                IF _sut_A._Step(_totalStepNumber - 1, TRUE, CONCAT('Step ', INT_TO_STRING(_totalStepNumber - 1))) THEN
                    _sut_A._SequenceComplete();
                END_IF

                _sut_A.SequencerClose();
                _sut_N.SequencerOpen();

                IF _sut_N._Step(0, TRUE, 'Step 0') THEN
                    _sut_N._StepCompleteWhen(TRUE);
                END_IF

                FOR i := 1 TO _totalStepNumber - 2 DO
                    _sut_N._Step(i, TRUE, CONCAT('Step ', INT_TO_STRING(i)));
                END_FOR

                IF _sut_N._Step(_totalStepNumber - 1, TRUE, CONCAT('Step ', INT_TO_STRING(_totalStepNumber - 1))) THEN
                    _sut_N._SequenceComplete();
                END_IF

                _sut_N.SequencerClose();
            END_IF

            IF _plcCycleCounter = 2 THEN
                _sut_A.SequencerOpen();

                IF _sut_A._Step(0, TRUE, 'Step 0') THEN
                    _sut_A._StepCompleteWhen(TRUE);
                END_IF

                IF _sut_A._Step(1, FALSE, 'Step 0') THEN
                    _sut_A._StepCompleteWhen(FALSE);
                END_IF

                _sut_N.SequencerOpen();

                IF _sut_N._Step(0, TRUE, 'Step 0') THEN
                    _sut_N._StepCompleteWhen(TRUE);
                END_IF

                IF _sut_N._Step(1, FALSE, 'Step 0') THEN
                    _sut_N._StepCompleteWhen(FALSE);
                END_IF
            END_IF

            IF _plcCycleCounter = 3 THEN
                FOR i := 2 TO _totalStepNumber - 1 DO
                    _sut_A._Step(i, TRUE, CONCAT('Step ', INT_TO_STRING(i)));
                END_FOR

                IF _sut_A._Step(_totalStepNumber, TRUE, CONCAT('Step ', INT_TO_STRING(_totalStepNumber))) THEN
                    _sut_A._SequenceComplete();
                END_IF

                _sut_A.SequencerClose();

                FOR i := 2 TO _totalStepNumber - 1 DO
                    _sut_N._Step(i, TRUE, CONCAT('Step ', INT_TO_STRING(i)));
                END_FOR

                IF _sut_N._Step(_totalStepNumber, TRUE, CONCAT('Step ', INT_TO_STRING(_totalStepNumber))) THEN
                    _sut_N._SequenceComplete();
                END_IF

                _sut_N.SequencerClose();
            END_IF

            _sut_A.SaveNumberOfStepsInSequence();
            _sut_N.SaveNumberOfStepsInSequence();
        END_IF

        _done := _plcCycleCounter >= 3;
        ProbeDoneWhen(_done);
        {endregion}
        {region "T560_RequestStepCallingCyclically"}
    eTcoSequencerTests.RequestStepCallingCyclically:
        IF NOT _arranged THEN
            _sut_A.TcoSequencerTest := eTcoSequencerTests.RequestStepCallingCyclically;
            _sut_N.TcoSequencerTest := eTcoSequencerTests.RequestStepCallingCyclically;
            _sut_A.SetCyclicMode(); //Set sequencer into the cyclic mode
            _sut_N.SetCyclicMode(); //Set sequencer into the cyclic mode
            _sut_A.SetSequenceAsChecked(); //Set sequence as checked, so no StepID uniqueness is performed on next sequence execution
            _sut_N.SetSequenceAsChecked(); //Set sequence as checked, so no StepID uniqueness is performed on next sequence execution
            _sut_A.SetNumberOfSteps(_totalStepNumber);
            _sut_N.SetNumberOfSteps(_totalStepNumber);
            _sut_A.TotalStepNumber := _totalStepNumber;
            _sut_N.TotalStepNumber := _totalStepNumber;
            _sut_A.InitReqStepCycle := _initReqStepCycle;
            _sut_N.InitReqStepCycle := _initReqStepCycle;
            _sut_A.SaveNumberOfStepsInSequence();
            _sut_N.SaveNumberOfStepsInSequence();
            _plcCycleCounter := 0;
            _arranged := TRUE;
            RETURN;
        END_IF

        IF NOT _done THEN
            IF _plcCycleCounter = 1 THEN
                _sut_A.SequencerOpen();
                _sut_N.SequencerOpen();
            END_IF

            IF _plcCycleCounter = 2 THEN
                _sut_A.SequencerOpen();
                _sut_A._RequestStep(10);
                _sut_A.SequencerClose();
                _sut_A.SequencerOpen();
                _sut_N.SequencerOpen();
                _sut_N._RequestStep(10);
                _sut_N.SequencerClose();
                _sut_N.SequencerOpen();
            END_IF

            IF _plcCycleCounter = 3 THEN
                _sut_A._Step(0, TRUE, 'Step 0');
                _sut_A._Step(20, TRUE, 'Step 20');
                _sut_A._Step(10, TRUE, 'Step 10');
                _sut_A.SequencerClose();
                _sut_N._Step(0, TRUE, 'Step 0');
                _sut_N._Step(20, TRUE, 'Step 20');
                _sut_N._Step(10, TRUE, 'Step 10');
                _sut_N.SequencerClose();
            END_IF

            IF _plcCycleCounter = 4 THEN
                _sut_A.InitReqStepCycle := _initReqStepCycle;
                _sut_N.InitReqStepCycle := _initReqStepCycle;
            END_IF

            IF _plcCycleCounter >= 5 THEN
                _sut_A.SequencerOpen();
                _sut_A.PostOpenRequestStepCycle := _sut_A.RequestStepCycle;
                _sut_A._Step(0, TRUE, 'Step 0');

                IF (_sut_A._Step(20, TRUE, 'Step 20')) THEN
                    _sut_A._RequestStep(20);
                END_IF

                IF (_sut_A._Step(10, TRUE, 'Step 10')) THEN
                    _sut_A._RequestStep(20);
                END_IF

                _sut_A.PreCloseRequestStepCycle := _sut_A.RequestStepCycle;
                _sut_A.SequencerClose();
                _sut_N.SequencerOpen();
                _sut_N.PostOpenRequestStepCycle := _sut_N.RequestStepCycle;
                _sut_N._Step(0, TRUE, 'Step 0');

                IF (_sut_N._Step(20, TRUE, 'Step 20')) THEN
                    _sut_N._RequestStep(20);
                END_IF

                IF (_sut_N._Step(10, TRUE, 'Step 10')) THEN
                    _sut_N._RequestStep(20);
                END_IF

                _sut_N.PreCloseRequestStepCycle := _sut_N.RequestStepCycle;
                _sut_N.SequencerClose();
            END_IF
        END_IF

        _sut_A.SaveNumberOfStepsInSequence();
        _sut_N.SaveNumberOfStepsInSequence();
        _done := _plcCycleCounter >= _cycles + 4;
        ProbeDoneWhen(_done);
        {endregion}
        {region "T570_SetStepMode"}
    eTcoSequencerTests.SetStepMode:
        IF NOT _arranged THEN
            _sut_A.TcoSequencerTest := eTcoSequencerTests.SetStepMode;
            _sut_N.TcoSequencerTest := eTcoSequencerTests.SetStepMode;
            _sut_A.SetStepMode(); //Set sequencer into the step mode
            _sut_N.SetStepMode(); //Set sequencer into the step mode
            _sut_A.SetSequenceAsChecked(); //Set sequence as checked, so no StepID uniqueness is performed on next sequence execution
            _sut_N.SetSequenceAsChecked(); //Set sequence as checked, so no StepID uniqueness is performed on next sequence execution
            _sut_A.ClearNumberOfSteps();
            _sut_N.ClearNumberOfSteps();
            _sut_A.SetCurrentStep(inStepID := _currentStepId, inStepDescription := _currentStepDescription);
            _sut_N.SetCurrentStep(inStepID := _currentStepId, inStepDescription := _currentStepDescription);
            _sut_A.TotalStepNumber := _totalStepNumber;
            _sut_N.TotalStepNumber := _totalStepNumber;
            _sut_A.SaveNumberOfStepsInSequence();
            _sut_N.SaveNumberOfStepsInSequence();
            _plcCycleCounter := 0;
            _arranged := TRUE;
            RETURN;
        END_IF

        IF NOT _done THEN
            _sut_A.SequenceRun := _plcCycleCounter;
            _sut_N.SequenceRun := _plcCycleCounter;

            IF _plcCycleCounter = 1 THEN
                _sut_A.Run();
                _sut_N.Run();
            END_IF

            IF _plcCycleCounter = 2 THEN
                _sut_A.SequencerOpen();
                _sut_A._StepIn();

                IF _sut_A._Step(0, TRUE, 'Initial step') THEN
                    _sut_A._StepCompleteWhen(TRUE);
                END_IF

                _sut_N.SequencerOpen();
                _sut_N._StepIn();

                IF _sut_N._Step(0, TRUE, 'Initial step') THEN
                    _sut_N._StepCompleteWhen(TRUE);
                END_IF
            END_IF

            IF _plcCycleCounter = 3 THEN
                IF _sut_A._Step(1, TRUE, 'Step 1') THEN
                    _sut_A._StepCompleteWhen(TRUE);
                END_IF

                IF _sut_N._Step(1, TRUE, 'Step 1') THEN
                    _sut_N._StepCompleteWhen(TRUE);
                END_IF

                FOR i := 2 TO _totalStepNumber - 2 DO
                    _sut_A._Step(i, TRUE, CONCAT('Step ', INT_TO_STRING(i)));
                    _sut_N._Step(i, TRUE, CONCAT('Step ', INT_TO_STRING(i)));
                END_FOR

                IF _sut_A._Step(_totalStepNumber - 1, TRUE, CONCAT('Step ', INT_TO_STRING(_totalStepNumber - 1))) THEN
                    _sut_A._SequenceComplete();
                END_IF

                IF _sut_N._Step(_totalStepNumber - 1, TRUE, CONCAT('Step ', INT_TO_STRING(_totalStepNumber - 1))) THEN
                    _sut_N._SequenceComplete();
                END_IF
            END_IF

            IF _plcCycleCounter = 4 THEN
                _sut_A.Run();
                _sut_N.Run();
            END_IF

            _sut_A.SaveNumberOfStepsInSequence();
            _sut_N.SaveNumberOfStepsInSequence();
        END_IF

        _done := _plcCycleCounter >= 4;
        ProbeDoneWhen(_done);
        {endregion}
        {region "T580_StepMode"}
    eTcoSequencerTests.StepMode:
        IF NOT _arranged THEN
            _sut_A.TcoSequencerTest := eTcoSequencerTests.StepMode;
            _sut_N.TcoSequencerTest := eTcoSequencerTests.StepMode;
            _sut_A.SetStepMode(); //Set sequencer into the step mode
            _sut_N.SetStepMode(); //Set sequencer into the step mode
            _sut_A.SetSequenceAsChecked(); //Set sequence as checked, so no StepID uniqueness is performed on next sequence execution
            _sut_N.SetSequenceAsChecked(); //Set sequence as checked, so no StepID uniqueness is performed on next sequence execution
            _sut_A.ClearNumberOfSteps();
            _sut_N.ClearNumberOfSteps();
            _sut_A.SetCurrentStep(inStepID := _currentStepId, inStepDescription := _currentStepDescription);
            _sut_N.SetCurrentStep(inStepID := _currentStepId, inStepDescription := _currentStepDescription);
            _sut_A.TotalStepNumber := _totalStepNumber;
            _sut_N.TotalStepNumber := _totalStepNumber;
            _sut_A.SaveNumberOfStepsInSequence();
            _sut_N.SaveNumberOfStepsInSequence();
            _plcCycleCounter := 0;
            _arranged := TRUE;
            RETURN;
        END_IF

        IF NOT _done THEN
            _sut_A.SequenceRun := _plcCycleCounter;
            _sut_N.SequenceRun := _plcCycleCounter;
            _sut_A.Run();
            _sut_N.Run();
            _sut_A.SaveNumberOfStepsInSequence();
            _sut_N.SaveNumberOfStepsInSequence();
        END_IF

        _done := _plcCycleCounter >= _totalStepNumber + 1;
        ProbeDoneWhen(_done);
        {endregion}
        {region "T582_InvalidMode"}
    eTcoSequencerTests.InvalidMode:
        IF NOT _arranged THEN
            _sut_A.TcoSequencerTest := eTcoSequencerTests.SetStepMode;
            _sut_N.TcoSequencerTest := eTcoSequencerTests.SetStepMode;
            _sut_A.SetCyclicMode(); //Set sequencer into the cyclic mode
            _sut_N.SetCyclicMode(); //Set sequencer into the cyclic mode
            _sut_A.SetSequenceAsChecked(); //Set sequence as checked, so no StepID uniqueness is performed on next sequence execution
            _sut_N.SetSequenceAsChecked(); //Set sequence as checked, so no StepID uniqueness is performed on next sequence execution
            _sut_A.SetNumberOfSteps(_totalStepNumber);
            _sut_N.SetNumberOfSteps(_totalStepNumber);
            _sut_A.SetCurrentStep(inStepID := _currentStepId, inStepDescription := _currentStepDescription);
            _sut_N.SetCurrentStep(inStepID := _currentStepId, inStepDescription := _currentStepDescription);
            _sut_A.TotalStepNumber := _totalStepNumber;
            _sut_N.TotalStepNumber := _totalStepNumber;
            _sut_A.SaveNumberOfStepsInSequence();
            _sut_N.SaveNumberOfStepsInSequence();
            _plcCycleCounter := 0;
            _arranged := TRUE;
            RETURN;
        END_IF

        IF NOT _done THEN
            _sut_A.SequenceRun := _plcCycleCounter;
            _sut_N.SequenceRun := _plcCycleCounter;

            IF _plcCycleCounter = 1 THEN
                _sut_A.SequencerOpen();
                _sut_N.SequencerOpen();

                FOR i := 0 TO _totalStepNumber - 1 DO
                    IF _sut_A._Step(i, TRUE, CONCAT('Step ', INT_TO_STRING(i))) THEN
                        _sut_A._StepCompleteWhen(TRUE);
                    END_IF

                    IF _sut_N._Step(i, TRUE, CONCAT('Step ', INT_TO_STRING(i))) THEN
                        _sut_N._StepCompleteWhen(TRUE);
                    END_IF
                END_FOR
            END_IF

            IF _plcCycleCounter = 2 THEN
                _sut_A._Step(_totalStepNumber, TRUE, CONCAT('Step ', INT_TO_STRING(_totalStepNumber)));
                _sut_N._Step(_totalStepNumber, TRUE, CONCAT('Step ', INT_TO_STRING(_totalStepNumber)));
                _sut_A.SequencerClose();
                _sut_N.SequencerClose();
            END_IF

            IF _plcCycleCounter = 3 THEN
                _sut_A.SequencerOpen();
                _sut_N.SequencerOpen();

                FOR i := 0 TO _totalStepNumber DO
                    _sut_A._Step(i, TRUE, CONCAT('Step ', INT_TO_STRING(i)));
                    _sut_N._Step(i, TRUE, CONCAT('Step ', INT_TO_STRING(i)));
                END_FOR

                _sut_A.SequencerClose();
                _sut_N.SequencerClose();
            END_IF

            _sut_A.SaveNumberOfStepsInSequence();
            _sut_N.SaveNumberOfStepsInSequence();
        END_IF

        _done := _plcCycleCounter >= 3;
        ProbeDoneWhen(_done);
        {endregion}
        {region "T582_StepInError"}
    eTcoSequencerTests.StepInError:
        IF NOT _arranged THEN
            _sut_A.TcoSequencerTest := eTcoSequencerTests.StepInError;
            _sut_N.TcoSequencerTest := eTcoSequencerTests.StepInError;
            _sut_A.SetCyclicMode(); //Set sequencer into the cyclic mode
            _sut_N.SetCyclicMode(); //Set sequencer into the cyclic mode
            _sut_A.SetSequenceAsChecked(); //Set sequence as checked, so no StepID uniqueness is performed on next sequence execution
            _sut_N.SetSequenceAsChecked(); //Set sequence as checked, so no StepID uniqueness is performed on next sequence execution
            _sut_A.SetNumberOfSteps(_totalStepNumber);
            _sut_N.SetNumberOfSteps(_totalStepNumber);
            _sut_A.SetCurrentStep(inStepID := _currentStepId, inStepDescription := _currentStepDescription);
            _sut_N.SetCurrentStep(inStepID := _currentStepId, inStepDescription := _currentStepDescription);
            _sut_A.TotalStepNumber := _totalStepNumber;
            _sut_N.TotalStepNumber := _totalStepNumber;
            _sut_A.SaveNumberOfStepsInSequence();
            _sut_N.SaveNumberOfStepsInSequence();
            _plcCycleCounter := 0;
            _arranged := TRUE;
            RETURN;
        END_IF

        IF NOT _done THEN
            _sut_A.SequenceRun := _plcCycleCounter;
            _sut_N.SequenceRun := _plcCycleCounter;

            IF _plcCycleCounter = 1 THEN
                _sut_A.SequencerOpen();
                _sut_N.SequencerOpen();

                FOR i := 0 TO _totalStepNumber - 1 DO
                    IF _sut_A._Step(i, TRUE, CONCAT('Step ', INT_TO_STRING(i))) THEN
                        _sut_A._StepCompleteWhen(TRUE);
                    END_IF

                    IF _sut_N._Step(i, TRUE, CONCAT('Step ', INT_TO_STRING(i))) THEN
                        _sut_N._StepCompleteWhen(TRUE);
                    END_IF
                END_FOR
            END_IF

            IF _plcCycleCounter = 2 THEN
                _sut_A._Step(_totalStepNumber, TRUE, CONCAT('Step ', INT_TO_STRING(_totalStepNumber)));
                _sut_N._Step(_totalStepNumber, TRUE, CONCAT('Step ', INT_TO_STRING(_totalStepNumber)));
                _sut_A.SequencerClose();
                _sut_N.SequencerClose();
            END_IF

            IF _plcCycleCounter = 3 THEN
                _sut_A.SequencerOpen();
                _sut_N.SequencerOpen();

                FOR i := 0 TO _totalStepNumber DO
                    _sut_A._Step(i, TRUE, CONCAT('Step ', INT_TO_STRING(i)));
                    _sut_N._Step(i, TRUE, CONCAT('Step ', INT_TO_STRING(i)));
                END_FOR

                _sut_A.SequencerClose();
                _sut_N.SequencerClose();
            END_IF

            _sut_A.SaveNumberOfStepsInSequence();
            _sut_N.SaveNumberOfStepsInSequence();
        END_IF

        _done := _plcCycleCounter >= 3;
        ProbeDoneWhen(_done);
        {endregion}
        {region "T590_CheckStepIdUniquenessStepMode"}
    eTcoSequencerTests.CheckStepIdUniquenessStepMode:
        IF NOT _arranged THEN
            _sut_A.SetStepMode(); //Set sequencer into the step mode
            _sut_N.SetStepMode(); //Set sequencer into the step mode
            _sut_A.SetSequenceAsNotChecked(); //Set sequence as not checked, so StepId uniqueness is going to be performed on next sequence run
            _sut_N.SetSequenceAsNotChecked(); //Set sequence as not checked, so StepId uniqueness is going to be performed on next sequence run
            _sut_A.ClearNumberOfSteps(); //Clear internal step counters, so number of steps is going to be counted again on next sequence run
            _sut_N.ClearNumberOfSteps(); //Clear internal step counters, so number of steps is going to be counted again on next sequence run
            _sut_A.Enabled := TRUE;
            _sut_A.RunOneStep := FALSE;
            _sut_A.RunAllSteps := TRUE;
            _sut_A.FinishStep := TRUE;
            _sut_A.StepId := _stepId;
            _sut_A.StepDescription := _stepDescription;
            _sut_N.Enabled := TRUE;
            _sut_N.RunOneStep := FALSE;
            _sut_N.RunAllSteps := TRUE;
            _sut_N.FinishStep := TRUE;
            _sut_N.StepId := _stepId;
            _sut_N.StepDescription := _stepDescription;
            _sut_A.SetCurrentStep(inStepID := _currentStepId, inStepDescription := _currentStepDescription);
            _sut_N.SetCurrentStep(inStepID := _currentStepId, inStepDescription := _currentStepDescription);
            _sut_A.TcoSequencerTest := eTcoSequencerTests.CheckStepIdUniquenessStepMode;
            _sut_N.TcoSequencerTest := eTcoSequencerTests.CheckStepIdUniquenessStepMode;
            _sut_A.SaveNumberOfStepsInSequence();
            _sut_N.SaveNumberOfStepsInSequence();
            _plcCycleCounter := 0;
            _arranged := TRUE;
            RETURN;
        END_IF

        IF NOT _done THEN
            IF _plcCycleCounter = 3 THEN
                _sut_A._StepIn();
                _sut_N._StepIn();
            END_IF

            _sut_A.Run();
            _sut_N.Run();

            IF _plcCycleCounter = 4 THEN
                _sut_A.Restore();
                _sut_N.Restore();
            END_IF

            _sut_A.SaveNumberOfStepsInSequence();
            _sut_N.SaveNumberOfStepsInSequence();
        END_IF

        _done := _plcCycleCounter >= 4;

        IF _done THEN
            _sut_A.TcoSequencerTest := eTcoSequencerTests.none;
            _sut_N.TcoSequencerTest := eTcoSequencerTests.none;
        END_IF

        ProbeDoneWhen(_done);
        {endregion}
        {region "T594_NotUniqueStepIdInStepMode"}
    eTcoSequencerTests.NotUniqueStepIdInStepMode:
        IF NOT _arranged THEN
            _sut_A.TcoSequencerTest := eTcoSequencerTests.NotUniqueStepIdInStepMode;
            _sut_N.TcoSequencerTest := eTcoSequencerTests.NotUniqueStepIdInStepMode;
            _sut_A.SetStepMode(); //Set sequencer into the step mode
            _sut_N.SetStepMode(); //Set sequencer into the step mode
            _sut_A.Enabled := TRUE;
            _sut_A.RunOneStep := FALSE;
            _sut_A.RunAllSteps := FALSE;
            _sut_A.FinishStep := TRUE;
            _sut_A.StepId := _stepId;
            _sut_N.Enabled := TRUE;
            _sut_N.RunOneStep := FALSE;
            _sut_N.RunAllSteps := FALSE;
            _sut_N.FinishStep := TRUE;
            _sut_N.StepId := _stepId;
            _sut_A.SetCurrentStep(inStepID := _currentStepId, inStepDescription := _currentStepDescription);
            _sut_N.SetCurrentStep(inStepID := _currentStepId, inStepDescription := _currentStepDescription);
            _sut_A.SaveNumberOfStepsInSequence();
            _sut_N.SaveNumberOfStepsInSequence();
            _plcCycleCounter := 0;
            _arranged := TRUE;
            RETURN;
        END_IF

        IF NOT _done THEN
            IF _plcCycleCounter = 2 THEN
                _Sut_A.RunOneStep := TRUE;
                _Sut_N.RunOneStep := TRUE;
            END_IF

            _sut_A.Run();
            _sut_N.Run();
            _sut_A.SaveNumberOfStepsInSequence();
            _sut_N.SaveNumberOfStepsInSequence();
            _done := _plcCycleCounter >= 2;
        END_IF

        IF _done THEN
            ProbeDoneWhen(_done);
        END_IF
        {endregion}
        {region "T597_AfterErrorResetInStepMode"}
    eTcoSequencerTests.AfterErrorResetInStepMode:
        IF NOT _arranged THEN
            _sut_A.TcoSequencerTest := eTcoSequencerTests.AfterErrorRestore;
            _sut_N.TcoSequencerTest := eTcoSequencerTests.AfterErrorRestore;
            _sut_A.SetStepMode();
            _sut_N.SetStepMode();
            _sut_A.SaveNumberOfStepsInSequence();
            _sut_N.SaveNumberOfStepsInSequence();
            _plcCycleCounter := 0;
            _arranged := TRUE;
            RETURN;
        END_IF

        IF NOT _done THEN
            IF _plcCycleCounter = 3 THEN
                _sut_A._StepIn();
                _sut_N._StepIn();
            END_IF

            _sut_A.Run();
            _sut_N.Run();
            _sut_A.SaveNumberOfStepsInSequence();
            _sut_N.SaveNumberOfStepsInSequence();
            _done := _plcCycleCounter >= 4;
        END_IF

        IF _done THEN
            ProbeDoneWhen(_done);
        END_IF
        {endregion}
        {region "T601_InvalidModeDetailed"}
    eTcoSequencerTests.InvalidModeDetailed:
        IF NOT _arranged THEN
            _sut_A.TcoSequencerTest := eTcoSequencerTests.InvalidModeDetailed;
            _sut_N.TcoSequencerTest := eTcoSequencerTests.InvalidModeDetailed;
            _sut_A.SetSequenceAsNotChecked();
            _sut_N.SetSequenceAsNotChecked();
            _sut_A.ClearNumberOfSteps();
            _sut_N.ClearNumberOfSteps();
            _sut_A.SetCurrentStep(_currentStepId, _currentStepDescription);
            _sut_N.SetCurrentStep(_currentStepId, _currentStepDescription);
            _sut_A.StepId := _stepId;
            _sut_N.StepId := _stepId;
            _sut_A.StepDescription := _stepDescription;
            _sut_N.StepDescription := _stepDescription;
            _sut_A.Enabled := TRUE;
            _sut_N.Enabled := TRUE;
            _sut_A.RunOneStep := FALSE;
            _sut_N.RunOneStep := FALSE;
            _sut_A.RunAllSteps := TRUE;
            _sut_N.RunAllSteps := TRUE;
            _sut_A.FinishStep := TRUE;
            _sut_N.FinishStep := TRUE;
            _sut_A.SetStepMode();
            _sut_N.SetStepMode();
            _sut_A.SaveNumberOfStepsInSequence();
            _sut_N.SaveNumberOfStepsInSequence();
            _plcCycleCounter := 0;
            _arranged := TRUE;
            RETURN;
        END_IF

        IF NOT _done THEN
            IF _plcCycleCounter = 2 THEN
                _sut_A.SetInvalidMode();
                _sut_N.SetInvalidMode();
                _sut_A.RunOneStep := TRUE;
                _sut_N.RunOneStep := TRUE;
                _sut_A.RunAllSteps := FALSE;
                _sut_N.RunAllSteps := FALSE;
            END_IF

            _sut_A.Run();
            _sut_N.Run();
            _sut_A.SaveNumberOfStepsInSequence();
            _sut_N.SaveNumberOfStepsInSequence();
            _done := _plcCycleCounter >= 2;
        END_IF

        IF _done THEN
            ProbeDoneWhen(_done);
        END_IF
        {endregion}
        {region "T604_StepInErrorDetailed"}
    eTcoSequencerTests.StepInErrorDetailed:
        IF NOT _arranged THEN
            _sut_A.TcoSequencerTest := eTcoSequencerTests.StepInErrorDetailed;
            _sut_N.TcoSequencerTest := eTcoSequencerTests.StepInErrorDetailed;
            _sut_A.SetSequenceAsNotChecked();
            _sut_N.SetSequenceAsNotChecked();
            _sut_A.ClearNumberOfSteps();
            _sut_N.ClearNumberOfSteps();
            _sut_A.SetCurrentStep(_currentStepId, _currentStepDescription);
            _sut_N.SetCurrentStep(_currentStepId, _currentStepDescription);
            _sut_A.StepId := _stepId;
            _sut_N.StepId := _stepId;
            _sut_A.StepDescription := _stepDescription;
            _sut_N.StepDescription := _stepDescription;
            _sut_A.Enabled := TRUE;
            _sut_N.Enabled := TRUE;
            _sut_A.RunOneStep := FALSE;
            _sut_N.RunOneStep := FALSE;
            _sut_A.RunAllSteps := TRUE;
            _sut_N.RunAllSteps := TRUE;
            _sut_A.FinishStep := TRUE;
            _sut_N.FinishStep := TRUE;
            _sut_A.SetStepMode();
            _sut_N.SetStepMode();
            _sut_A.SaveNumberOfStepsInSequence();
            _sut_N.SaveNumberOfStepsInSequence();
            _plcCycleCounter := 0;
            _arranged := TRUE;
            RETURN;
        END_IF

        IF NOT _done THEN
            IF _plcCycleCounter = 2 THEN
                _sut_A.SetCurrentStepToErrorState();
                _sut_N.SetCurrentStepToErrorState();
                _sut_A.RunOneStep := TRUE;
                _sut_N.RunOneStep := TRUE;
                _sut_A.RunAllSteps := FALSE;
                _sut_N.RunAllSteps := FALSE;
            END_IF

            _sut_A.Run();
            _sut_N.Run();
            _sut_A.SaveNumberOfStepsInSequence();
            _sut_N.SaveNumberOfStepsInSequence();
            _done := _plcCycleCounter >= 2;
        END_IF

        IF _done THEN
            ProbeDoneWhen(_done);
        END_IF
        {endregion}
        {region "T611_StepModeStepIn"}
    eTcoSequencerTests.StepModeStepIn:
        IF NOT _arranged THEN
            _sut_A.TcoSequencerTest := eTcoSequencerTests.StepModeStepIn;
            _sut_N.TcoSequencerTest := eTcoSequencerTests.StepModeStepIn;
            _sut_A.SetSequenceAsChecked();
            _sut_N.SetSequenceAsChecked();
            _sut_A.SetNumberOfSteps(_totalStepNumber);
            _sut_N.SetNumberOfSteps(_totalStepNumber);
            _sut_A.TotalStepNumber := _totalStepNumber;
            _sut_N.TotalStepNumber := _totalStepNumber;
            _sut_A.SetCurrentStep(_currentStepId, _currentStepDescription);
            _sut_N.SetCurrentStep(_currentStepId, _currentStepDescription);
            _sut_A.StepId := _stepId;
            _sut_N.StepId := _stepId;
            _sut_A.StepDescription := _stepDescription;
            _sut_N.StepDescription := _stepDescription;
            _sut_A.Enabled := TRUE;
            _sut_N.Enabled := TRUE;
            _sut_A.RunOneStep := FALSE;
            _sut_N.RunOneStep := FALSE;
            _sut_A.RunAllSteps := TRUE;
            _sut_N.RunAllSteps := TRUE;
            _sut_A.FinishStep := TRUE;
            _sut_N.FinishStep := TRUE;
            _sut_A.SetStepMode();
            _sut_N.SetStepMode();
            _sut_A.SaveNumberOfStepsInSequence();
            _sut_N.SaveNumberOfStepsInSequence();
            _plcCycleCounter := 0;
            _arranged := TRUE;
            RETURN;
        END_IF

        IF NOT _done THEN
            _sut_A.SequenceRun := _plcCycleCounter;
            _sut_N.SequenceRun := _plcCycleCounter;
            _sut_A.Run();
            _sut_N.Run();
            _sut_A.SaveNumberOfStepsInSequence();
            _sut_N.SaveNumberOfStepsInSequence();
            _done := _plcCycleCounter >= _totalStepNumber + 1;
        END_IF

        IF _done THEN
            ProbeDoneWhen(_done);
        END_IF
        {endregion}
        {region "T612_StepModeChangeStepIdDuringExecution"}
    eTcoSequencerTests.StepModeChangeStepIdDuringExecution:
        IF NOT _done AND _plcCycleCounter <= 2 THEN
            _sut_A.TcoSequencerTest := eTcoSequencerTests.StepModeChangeStepIdDuringExecution;
            _sut_N.TcoSequencerTest := eTcoSequencerTests.StepModeChangeStepIdDuringExecution;
            _sut_A.SequenceRun := _plcCycleCounter;
            _sut_N.SequenceRun := _plcCycleCounter;
            _sut_A.Run();
            _sut_N.Run();
            _sut_A.SaveNumberOfStepsInSequence();
            _sut_N.SaveNumberOfStepsInSequence();
        END_IF

        IF _plcCycleCounter >= 3 THEN
            _sut_A.Restore();
            _sut_N.Restore();
            _sut_A.SetSequenceAsChecked();
            _sut_N.SetSequenceAsChecked();
            _sut_A.SetNumberOfSteps(_totalStepNumber);
            _sut_N.SetNumberOfSteps(_totalStepNumber);
            _sut_A.TotalStepNumber := _totalStepNumber;
            _sut_N.TotalStepNumber := _totalStepNumber;
            _sut_A.SetStepMode();
            _sut_N.SetStepMode();
            _sut_A.SaveNumberOfStepsInSequence();
            _sut_N.SaveNumberOfStepsInSequence();
        END_IF

        _done := _plcCycleCounter >= 3;

        IF _done THEN
            ProbeDoneWhen(_done);
        END_IF
        {endregion}
        {region "T615_StepModeChangeStepOrder"}
    eTcoSequencerTests.StepModeChangeStepOrder:
        IF NOT _arranged THEN
            _sut_A.TcoSequencerTest := eTcoSequencerTests.StepModeChangeStepOrder;
            _sut_N.TcoSequencerTest := eTcoSequencerTests.StepModeChangeStepOrder;
            _sut_A.SetSequenceAsChecked();
            _sut_N.SetSequenceAsChecked();
            _sut_A.SetNumberOfSteps(_totalStepNumber);
            _sut_N.SetNumberOfSteps(_totalStepNumber);
            _sut_A.TotalStepNumber := _totalStepNumber;
            _sut_N.TotalStepNumber := _totalStepNumber;
            _sut_A.SetCurrentStep(_currentStepId, _currentStepDescription);
            _sut_N.SetCurrentStep(_currentStepId, _currentStepDescription);
            _sut_A.StepId := _stepId;
            _sut_N.StepId := _stepId;
            _sut_A.StepDescription := _stepDescription;
            _sut_N.StepDescription := _stepDescription;
            _sut_A.Enabled := TRUE;
            _sut_N.Enabled := TRUE;
            _sut_A.RunOneStep := FALSE;
            _sut_N.RunOneStep := FALSE;
            _sut_A.RunAllSteps := TRUE;
            _sut_N.RunAllSteps := TRUE;
            _sut_A.FinishStep := TRUE;
            _sut_N.FinishStep := TRUE;
            _sut_A.SetStepMode();
            _sut_N.SetStepMode();
            _sut_A.SaveNumberOfStepsInSequence();
            _sut_N.SaveNumberOfStepsInSequence();
            _plcCycleCounter := 0;
            _arranged := TRUE;
            RETURN;
        END_IF

        IF _plcCycleCounter <= _totalStepNumber + 2 THEN
            _sut_A.SequenceRun := _plcCycleCounter;
            _sut_N.SequenceRun := _plcCycleCounter;
            _sut_A.Run();
            _sut_N.Run();
            _sut_A.SaveNumberOfStepsInSequence();
            _sut_N.SaveNumberOfStepsInSequence();
        END_IF

        IF _plcCycleCounter >= _totalStepNumber + 3 THEN
            _sut_A.Restore();
            _sut_N.Restore();
            _sut_A.SetSequenceAsChecked();
            _sut_N.SetSequenceAsChecked();
            _sut_A.SetNumberOfSteps(_totalStepNumber);
            _sut_N.SetNumberOfSteps(_totalStepNumber);
            _sut_A.TotalStepNumber := _totalStepNumber;
            _sut_N.TotalStepNumber := _totalStepNumber;
            _sut_A.SetStepMode();
            _sut_N.SetStepMode();
            _sut_A.SaveNumberOfStepsInSequence();
            _sut_N.SaveNumberOfStepsInSequence();
        END_IF

        _done := _plcCycleCounter >= _totalStepNumber + 3;

        IF _done THEN
            ProbeDoneWhen(_done);
        END_IF
        {endregion}
        {region "T618_StepModeCommentOutPartOfRunningSequencer"}
    eTcoSequencerTests.StepModeCommentOutPartOfRunningSequencer:
        IF NOT _arranged THEN
            _sut_A.TcoSequencerTest := eTcoSequencerTests.StepModeCommentOutPartOfRunningSequencer;
            _sut_N.TcoSequencerTest := eTcoSequencerTests.StepModeCommentOutPartOfRunningSequencer;
            _sut_A.SetStepMode(); //Set sequencer into the step mode
            _sut_N.SetStepMode(); //Set sequencer into the step mode
            _sut_A.SetSequenceAsChecked(); //Set sequence as checked, so no StepID uniqueness is performed on next sequence execution
            _sut_N.SetSequenceAsChecked(); //Set sequence as checked, so no StepID uniqueness is performed on next sequence execution
            _sut_A.ClearNumberOfSteps(); //Clear internal step counters, so number of steps is going to be counted again on next sequence run
            _sut_N.ClearNumberOfSteps(); //Clear internal step counters, so number of steps is going to be counted again on next sequence run
            _sut_A.SetCurrentStep(inStepID := _currentStepId, inStepDescription := _currentStepDescription);
            _sut_N.SetCurrentStep(inStepID := _currentStepId, inStepDescription := _currentStepDescription);
            _sut_A.TotalStepNumber := _totalStepNumber;
            _sut_N.TotalStepNumber := _totalStepNumber;
            _sut_A.SaveNumberOfStepsInSequence();
            _sut_N.SaveNumberOfStepsInSequence();
            _plcCycleCounter := 0;
            _arranged := TRUE;
            RETURN;
        END_IF

        IF NOT _done THEN
            IF _plcCycleCounter = 3 THEN
                _sut_A.Restore();
                _sut_N.Restore();
                _sut_A.SetSequenceAsChecked(); //Set sequence as checked, so no StepID uniqueness is performed on next sequence execution
                _sut_N.SetSequenceAsChecked(); //Set sequence as checked, so no StepID uniqueness is performed on next sequence execution
                _sut_A.ClearNumberOfSteps(); //Clear internal step counters, so number of steps is going to be counted again on next sequence run
                _sut_N.ClearNumberOfSteps(); //Clear internal step counters, so number of steps is going to be counted again on next sequence run
            END_IF

            _sut_A.SequenceRun := _plcCycleCounter;
            _sut_N.SequenceRun := _plcCycleCounter;
            _sut_A.Run();
            _sut_N.Run();
            _sut_A.SaveNumberOfStepsInSequence();
            _sut_N.SaveNumberOfStepsInSequence();
        END_IF

        _done := _plcCycleCounter >= 3;
        ProbeDoneWhen(_done);
        {endregion}
        {region "T621_StepModeUncommentPartOfRunningSequencer"}
    eTcoSequencerTests.StepModeUncommentPartOfRunningSequencer:
        IF NOT _arranged THEN
            _sut_A.TcoSequencerTest := eTcoSequencerTests.StepModeUncommentPartOfRunningSequencer;
            _sut_N.TcoSequencerTest := eTcoSequencerTests.StepModeUncommentPartOfRunningSequencer;
            _sut_A.SetStepMode(); //Set sequencer into the step mode
            _sut_N.SetStepMode(); //Set sequencer into the step mode
            _sut_A.SetSequenceAsChecked(); //Set sequence as checked, so no StepID uniqueness is performed on next sequence execution
            _sut_N.SetSequenceAsChecked(); //Set sequence as checked, so no StepID uniqueness is performed on next sequence execution
            _sut_A.ClearNumberOfSteps(); //Clear internal step counters, so number of steps is going to be counted again on next sequence run
            _sut_N.ClearNumberOfSteps(); //Clear internal step counters, so number of steps is going to be counted again on next sequence run
            _sut_A.SetCurrentStep(inStepID := _currentStepId, inStepDescription := _currentStepDescription);
            _sut_N.SetCurrentStep(inStepID := _currentStepId, inStepDescription := _currentStepDescription);
            _sut_A.TotalStepNumber := _totalStepNumber;
            _sut_N.TotalStepNumber := _totalStepNumber;
            _sut_A.SaveNumberOfStepsInSequence();
            _sut_N.SaveNumberOfStepsInSequence();
            _plcCycleCounter := 0;
            _arranged := TRUE;
            RETURN;
        END_IF

        IF NOT _done THEN
            _sut_A.SequenceRun := _plcCycleCounter;
            _sut_N.SequenceRun := _plcCycleCounter;
            _sut_A.Run();
            _sut_N.Run();
            _sut_A.SaveNumberOfStepsInSequence();
            _sut_N.SaveNumberOfStepsInSequence();
        END_IF

        _done := _plcCycleCounter >= 2;
        ProbeDoneWhen(_done);
        {endregion}
        {region "T631_StepModeRequestStepFromLowerToHigher"}
    eTcoSequencerTests.StepModeRequestStepFromLowerToHigher:
        IF NOT _arranged THEN
            _sut_A.TcoSequencerTest := eTcoSequencerTests.StepModeRequestStepFromLowerToHigher;
            _sut_N.TcoSequencerTest := eTcoSequencerTests.StepModeRequestStepFromLowerToHigher;
            _sut_A.SetStepMode(); //Set sequencer into the step mode
            _sut_N.SetStepMode(); //Set sequencer into the step mode
            _sut_A.SetSequenceAsChecked(); //Set sequence as checked, so no StepID uniqueness is performed on next sequence execution
            _sut_N.SetSequenceAsChecked(); //Set sequence as checked, so no StepID uniqueness is performed on next sequence execution
            _sut_A.ClearNumberOfSteps(); //Clear internal step counters, so number of steps is going to be counted again on next sequence run
            _sut_N.ClearNumberOfSteps(); //Clear internal step counters, so number of steps is going to be counted again on next sequence run
            _sut_A.SetCurrentStep(inStepID := _currentStepId, inStepDescription := _currentStepDescription);
            _sut_N.SetCurrentStep(inStepID := _currentStepId, inStepDescription := _currentStepDescription);
            _sut_A.TotalStepNumber := _totalStepNumber;
            _sut_N.TotalStepNumber := _totalStepNumber;
            _sut_A.ReqStep := _reqStep;
            _sut_N.ReqStep := _reqStep;
            _sut_A.ReqStepNotExists := _reqStepNotExists;
            _sut_N.ReqStepNotExists := _reqStepNotExists;
            _sut_A.SaveNumberOfStepsInSequence();
            _sut_N.SaveNumberOfStepsInSequence();
            _plcCycleCounter := 0;
            _arranged := TRUE;
            RETURN;
        END_IF

        IF NOT _done THEN
            _sut_A.SequenceRun := _plcCycleCounter;
            _sut_N.SequenceRun := _plcCycleCounter;
            _sut_A.Run();
            _sut_N.Run();
            _sut_A.SaveNumberOfStepsInSequence();
            _sut_N.SaveNumberOfStepsInSequence();
        END_IF

        _done := _plcCycleCounter >= 2;
        ProbeDoneWhen(_done);
        {endregion}
        {region "T633_StepModeRequestStepFromHigherToLower"}
    eTcoSequencerTests.StepModeRequestStepFromHigherToLower:
        IF NOT _arranged THEN
            _sut_A.TcoSequencerTest := eTcoSequencerTests.StepModeRequestStepFromHigherToLower;
            _sut_N.TcoSequencerTest := eTcoSequencerTests.StepModeRequestStepFromHigherToLower;
            _sut_A.SetStepMode(); //Set sequencer into the step mode
            _sut_N.SetStepMode(); //Set sequencer into the step mode
            _sut_A.SetSequenceAsChecked(); //Set sequence as checked, so no StepID uniqueness is performed on next sequence execution
            _sut_N.SetSequenceAsChecked(); //Set sequence as checked, so no StepID uniqueness is performed on next sequence execution
            _sut_A.SetNumberOfSteps(_totalStepNumber);
            _sut_N.SetNumberOfSteps(_totalStepNumber);
            _sut_A.SetCurrentStep(inStepID := _currentStepId, inStepDescription := _currentStepDescription);
            _sut_N.SetCurrentStep(inStepID := _currentStepId, inStepDescription := _currentStepDescription);
            _sut_A.TotalStepNumber := _totalStepNumber;
            _sut_N.TotalStepNumber := _totalStepNumber;
            _sut_A.ReqStep := _reqStep;
            _sut_N.ReqStep := _reqStep;
            _sut_A.ReqStepNotExists := _reqStepNotExists;
            _sut_N.ReqStepNotExists := _reqStepNotExists;
            _sut_A.SaveNumberOfStepsInSequence();
            _sut_N.SaveNumberOfStepsInSequence();
            _plcCycleCounter := 0;
            _arranged := TRUE;
            RETURN;
        END_IF

        IF NOT _done THEN
            _sut_A.SequenceRun := _plcCycleCounter;
            _sut_N.SequenceRun := _plcCycleCounter;
            _sut_A.Run();
            _sut_N.Run();
            _sut_A.SaveNumberOfStepsInSequence();
            _sut_N.SaveNumberOfStepsInSequence();
        END_IF

        _done := _plcCycleCounter >= _reqStep + 7;
        ProbeDoneWhen(_done);
        {endregion}
        {region "T635_StepModeRequestStepToNotExistingStep"}
    eTcoSequencerTests.StepModeRequestStepToNotExistingStep:
        IF NOT _arranged THEN
            _sut_A.TcoSequencerTest := eTcoSequencerTests.RequestStepToNotExistingStep;
            _sut_N.TcoSequencerTest := eTcoSequencerTests.RequestStepToNotExistingStep;
            _sut_A.SetStepMode(); //Set sequencer into the step mode
            _sut_N.SetStepMode(); //Set sequencer into the step mode
            _sut_A.SetSequenceAsChecked(); //Set sequence as checked, so no StepID uniqueness is performed on next sequence execution
            _sut_N.SetSequenceAsChecked(); //Set sequence as checked, so no StepID uniqueness is performed on next sequence execution
            _sut_A.SetNumberOfSteps(_totalStepNumber);
            _sut_N.SetNumberOfSteps(_totalStepNumber);
            _sut_A.SetCurrentStep(inStepID := _currentStepId, inStepDescription := _currentStepDescription);
            _sut_N.SetCurrentStep(inStepID := _currentStepId, inStepDescription := _currentStepDescription);
            _sut_A.TotalStepNumber := _totalStepNumber;
            _sut_N.TotalStepNumber := _totalStepNumber;
            _sut_A.ReqStep := _reqStep;
            _sut_N.ReqStep := _reqStep;
            _sut_A.ReqStepNotExists := _reqStepNotExists;
            _sut_N.ReqStepNotExists := _reqStepNotExists;
            _sut_A.SaveNumberOfStepsInSequence();
            _sut_N.SaveNumberOfStepsInSequence();
            _plcCycleCounter := 0;
            _arranged := TRUE;
            RETURN;
        END_IF

        IF _plcCycleCounter = 4 THEN
            _sut_A.Restore();
            _sut_N.Restore();
            _sut_A.SetStepMode(); //Set sequencer into the step mode
            _sut_N.SetStepMode(); //Set sequencer into the step mode
            _sut_A.SetSequenceAsChecked(); //Set sequence as checked, so no StepID uniqueness is performed on next sequence execution
            _sut_N.SetSequenceAsChecked(); //Set sequence as checked, so no StepID uniqueness is performed on next sequence execution
            _sut_A.SetNumberOfSteps(_totalStepNumber);
            _sut_N.SetNumberOfSteps(_totalStepNumber);
            _sut_A.SetCurrentStep(inStepID := _currentStepId, inStepDescription := _currentStepDescription);
            _sut_N.SetCurrentStep(inStepID := _currentStepId, inStepDescription := _currentStepDescription);
            _sut_A.TotalStepNumber := _totalStepNumber;
            _sut_N.TotalStepNumber := _totalStepNumber;
        END_IF

        IF NOT _done THEN
            _sut_A.SequenceRun := _plcCycleCounter;
            _sut_N.SequenceRun := _plcCycleCounter;
            _sut_A.Run();
            _sut_N.Run();
            _sut_A.SaveNumberOfStepsInSequence();
            _sut_N.SaveNumberOfStepsInSequence();
        END_IF

        _done := _plcCycleCounter >= 4;
        ProbeDoneWhen(_done);
        {endregion}
        {region "T640_StepModeRequestStepWhilePreviousRequestStepHasnotBeenYetProcessed"}
    eTcoSequencerTests.StepModeRequestStepWhilePreviousRequestStepHasnotBeenYetProcessed:
        IF NOT _arranged THEN
            _sut_A.TcoSequencerTest := eTcoSequencerTests.StepModeRequestStepWhilePreviousRequestStepHasnotBeenYetProcessed;
            _sut_N.TcoSequencerTest := eTcoSequencerTests.StepModeRequestStepWhilePreviousRequestStepHasnotBeenYetProcessed;
            _sut_A.SetStepMode(); //Set sequencer into the step mode
            _sut_N.SetStepMode(); //Set sequencer into the step mode
            _sut_A.SetSequenceAsChecked(); //Set sequence as checked, so no StepID uniqueness is performed on next sequence execution
            _sut_N.SetSequenceAsChecked(); //Set sequence as checked, so no StepID uniqueness is performed on next sequence execution
            _sut_A.SetNumberOfSteps(_totalStepNumber);
            _sut_N.SetNumberOfSteps(_totalStepNumber);
            _sut_A.SetCurrentStep(inStepID := _currentStepId, inStepDescription := _currentStepDescription);
            _sut_N.SetCurrentStep(inStepID := _currentStepId, inStepDescription := _currentStepDescription);
            _sut_A.TotalStepNumber := _totalStepNumber;
            _sut_N.TotalStepNumber := _totalStepNumber;
            _sut_A.ReqStep := _reqStep;
            _sut_N.ReqStep := _reqStep;
            _sut_A.ReqStepNotExists := _reqStepNotExists;
            _sut_N.ReqStepNotExists := _reqStepNotExists;
            _sut_A.SaveNumberOfStepsInSequence();
            _sut_N.SaveNumberOfStepsInSequence();
            _plcCycleCounter := 0;
            _arranged := TRUE;
            RETURN;
        END_IF

        IF NOT _done THEN
            _sut_A.SequenceRun := _plcCycleCounter;
            _sut_N.SequenceRun := _plcCycleCounter;
            _sut_A.Run();
            _sut_N.Run();
            _sut_A.SaveNumberOfStepsInSequence();
            _sut_N.SaveNumberOfStepsInSequence();
        END_IF

        _done := TRUE;
        ProbeDoneWhen(_done);
        {endregion}
        {region "T641_StepModeDisabledStep"}
    eTcoSequencerTests.StepModeDisabledStep:
        IF NOT _arranged THEN
            _sut_A.TcoSequencerTest := eTcoSequencerTests.StepModeDisabledStep;
            _sut_N.TcoSequencerTest := eTcoSequencerTests.StepModeDisabledStep;
            _sut_A.SetStepMode(); //Set sequencer into the step mode
            _sut_N.SetStepMode(); //Set sequencer into the step mode
            _sut_A.SetSequenceAsChecked(); //Set sequence as checked, so no StepID uniqueness is performed on next sequence execution
            _sut_N.SetSequenceAsChecked(); //Set sequence as checked, so no StepID uniqueness is performed on next sequence execution
            _sut_A.SetNumberOfSteps(_totalStepNumber);
            _sut_N.SetNumberOfSteps(_totalStepNumber);
            _sut_A.TotalStepNumber := _totalStepNumber;
            _sut_N.TotalStepNumber := _totalStepNumber;
            _sut_A.SaveNumberOfStepsInSequence();
            _sut_N.SaveNumberOfStepsInSequence();
            _plcCycleCounter := 0;
            _arranged := TRUE;
            RETURN;
        END_IF

        IF NOT _done THEN
            _sut_A.SequenceRun := _plcCycleCounter;
            _sut_N.SequenceRun := _plcCycleCounter;
            _sut_A.Run();
            _sut_N.Run();
            _sut_A.SaveNumberOfStepsInSequence();
            _sut_N.SaveNumberOfStepsInSequence();
        END_IF

        _done := _plcCycleCounter >= 6;
        ProbeDoneWhen(_done);
        {endregion}
        {region "T670_StepModeStepForwardBackward"}
    eTcoSequencerTests.StepModeStepForwardBackward:
        IF NOT _arranged THEN
            _sut_A.TcoSequencerTest := eTcoSequencerTests.StepModeStepForwardBackward;
            _sut_N.TcoSequencerTest := eTcoSequencerTests.StepModeStepForwardBackward;
            _sut_A.SetStepMode(); //Set sequencer into the step mode
            _sut_N.SetStepMode(); //Set sequencer into the step mode
            _sut_A.SetSequenceAsChecked(); //Set sequence as checked, so no StepID uniqueness is performed on next sequence execution
            _sut_N.SetSequenceAsChecked(); //Set sequence as checked, so no StepID uniqueness is performed on next sequence execution
            _sut_A.SetNumberOfSteps(_totalStepNumber);
            _sut_N.SetNumberOfSteps(_totalStepNumber);
            _sut_A.TotalStepNumber := _totalStepNumber;
            _sut_N.TotalStepNumber := _totalStepNumber;
            _sut_A.SaveNumberOfStepsInSequence();
            _sut_N.SaveNumberOfStepsInSequence();
            _plcCycleCounter := 0;
            _arranged := TRUE;
            RETURN;
        END_IF

        IF NOT _done THEN
            _sut_A.SequenceRun := _plcCycleCounter;
            _sut_N.SequenceRun := _plcCycleCounter;
            _sut_A.Run();
            _sut_N.Run();
            _sut_A.SaveNumberOfStepsInSequence();
            _sut_N.SaveNumberOfStepsInSequence();
        END_IF

        _done := _plcCycleCounter >= 9;
        ProbeDoneWhen(_done);
        {endregion}
        {region "T681_StepModeStepInDetailed"}
    eTcoSequencerTests.StepModeStepInDetailed:
        IF NOT _arranged THEN
            _sut_A.TcoSequencerTest := eTcoSequencerTests.StepModeStepInDetailed;
            _sut_N.TcoSequencerTest := eTcoSequencerTests.StepModeStepInDetailed;
            _sut_A.SetStepMode(); //Set sequencer into the step mode
            _sut_N.SetStepMode(); //Set sequencer into the step mode
            _sut_A.SetSequenceAsChecked(); //Set sequence as checked, so no StepID uniqueness is performed on next sequence execution
            _sut_N.SetSequenceAsChecked(); //Set sequence as checked, so no StepID uniqueness is performed on next sequence execution
            _sut_A.SetNumberOfSteps(_totalStepNumber);
            _sut_N.SetNumberOfSteps(_totalStepNumber);
            _sut_A.TotalStepNumber := _totalStepNumber;
            _sut_N.TotalStepNumber := _totalStepNumber;
            _sut_A.SaveNumberOfStepsInSequence();
            _sut_N.SaveNumberOfStepsInSequence();
            _plcCycleCounter := 0;
            _arranged := TRUE;
            RETURN;
        END_IF

        IF NOT _done THEN
            _sut_A.SequenceRun := _plcCycleCounter;
            _sut_N.SequenceRun := _plcCycleCounter;
            _sut_A.Run();
            _sut_N.Run();
            _sut_A.SaveNumberOfStepsInSequence();
            _sut_N.SaveNumberOfStepsInSequence();
        END_IF

        _done := _plcCycleCounter >= 5;
        ProbeDoneWhen(_done);
        {endregion}
        {region "T691_SwitchStepModeOnDuringStepExecution"}
    eTcoSequencerTests.SwitchStepModeOnDuringStepExecution:
        IF NOT _arranged THEN
            _sut_A.TcoSequencerTest := eTcoSequencerTests.SwitchStepModeOnDuringStepExecution;
            _sut_N.TcoSequencerTest := eTcoSequencerTests.SwitchStepModeOnDuringStepExecution;
            _sut_A.SetCyclicMode(); //Set sequencer into the cyclic mode
            _sut_N.SetCyclicMode(); //Set sequencer into the cyclic mode
            _sut_A.SetSequenceAsChecked(); //Set sequence as checked, so no StepID uniqueness is performed on next sequence execution
            _sut_N.SetSequenceAsChecked(); //Set sequence as checked, so no StepID uniqueness is performed on next sequence execution
            _sut_A.SetNumberOfSteps(_totalStepNumber);
            _sut_N.SetNumberOfSteps(_totalStepNumber);
            _sut_A.TotalStepNumber := _totalStepNumber;
            _sut_N.TotalStepNumber := _totalStepNumber;
            _sut_A.SaveNumberOfStepsInSequence();
            _sut_N.SaveNumberOfStepsInSequence();
            _plcCycleCounter := 0;
            _arranged := TRUE;
            RETURN;
        END_IF

        IF NOT _done THEN
            _sut_A.SequenceRun := _plcCycleCounter;
            _sut_N.SequenceRun := _plcCycleCounter;
            _sut_A.Run();
            _sut_N.Run();
            _sut_A.SaveNumberOfStepsInSequence();
            _sut_N.SaveNumberOfStepsInSequence();
        END_IF

        _done := _plcCycleCounter >= 10;
        ProbeDoneWhen(_done);
        {endregion}
        {region "T693_SwitchStepModeStepForwardFromRunningStep"}
    eTcoSequencerTests.StepModeStepForwardFromRunningStep:
        _sut_A.TcoSequencerTest := eTcoSequencerTests.StepModeStepForwardFromRunningStep;
        _sut_N.TcoSequencerTest := eTcoSequencerTests.StepModeStepForwardFromRunningStep;

        IF NOT _done THEN
            _sut_A.SequenceRun := _plcCycleCounter;
            _sut_N.SequenceRun := _plcCycleCounter;
            _sut_A.Run();
            _sut_N.Run();
            _sut_A.SaveNumberOfStepsInSequence();
            _sut_N.SaveNumberOfStepsInSequence();
        END_IF

        _done := _plcCycleCounter >= 20;
        ProbeDoneWhen(_done);
        {endregion}
        {region "T695_SwitchStepModeStepBackwardFromRunningStep"}
    eTcoSequencerTests.StepModeStepBackwardFromRunningStep:
        _sut_A.TcoSequencerTest := eTcoSequencerTests.StepModeStepBackwardFromRunningStep;
        _sut_N.TcoSequencerTest := eTcoSequencerTests.StepModeStepBackwardFromRunningStep;

        IF NOT _done THEN
            _sut_A.SequenceRun := _plcCycleCounter;
            _sut_N.SequenceRun := _plcCycleCounter;
            _sut_A.Run();
            _sut_N.Run();
            _sut_A.SaveNumberOfStepsInSequence();
            _sut_N.SaveNumberOfStepsInSequence();
        END_IF

        _done := _plcCycleCounter >= 20;
        ProbeDoneWhen(_done);
        {endregion}
        {region "T696_SwitchStepModeStepOffFromReadyToRun"}
    eTcoSequencerTests.SwitchStepModeStepOffFromReadyToRun:
        _sut_A.TcoSequencerTest := eTcoSequencerTests.SwitchStepModeStepOffFromReadyToRun;
        _sut_N.TcoSequencerTest := eTcoSequencerTests.SwitchStepModeStepOffFromReadyToRun;

        IF NOT _done THEN
            _sut_A.SequenceRun := _plcCycleCounter;
            _sut_N.SequenceRun := _plcCycleCounter;
            _sut_A.Run();
            _sut_N.Run();
            _sut_A.SaveNumberOfStepsInSequence();
            _sut_N.SaveNumberOfStepsInSequence();
        END_IF

        _done := _plcCycleCounter >= 10;
        ProbeDoneWhen(_done);
        {endregion}
        {region "T697_SwitchStepModeStepOnFromRunning"}
    eTcoSequencerTests.SwitchStepModeStepOnFromRunning:
        _sut_A.TcoSequencerTest := eTcoSequencerTests.SwitchStepModeStepOnFromRunning;
        _sut_N.TcoSequencerTest := eTcoSequencerTests.SwitchStepModeStepOnFromRunning;

        IF NOT _done THEN
            _sut_A.SequenceRun := _plcCycleCounter;
            _sut_N.SequenceRun := _plcCycleCounter;
            _sut_A.Run();
            _sut_N.Run();
            _sut_A.SaveNumberOfStepsInSequence();
            _sut_N.SaveNumberOfStepsInSequence();
        END_IF

        _done := _plcCycleCounter >= 10;
        ProbeDoneWhen(_done);
        {endregion}
        {region "T698_SwitchStepModeStepOffFromRunning"}
    eTcoSequencerTests.SwitchStepModeStepOffFromRunning:
        _sut_A.TcoSequencerTest := eTcoSequencerTests.SwitchStepModeStepOffFromRunning;
        _sut_N.TcoSequencerTest := eTcoSequencerTests.SwitchStepModeStepOffFromRunning;

        IF NOT _done THEN
            _sut_A.SequenceRun := _plcCycleCounter;
            _sut_N.SequenceRun := _plcCycleCounter;
            _sut_A.Run();
            _sut_N.Run();
            _sut_A.SaveNumberOfStepsInSequence();
            _sut_N.SaveNumberOfStepsInSequence();
        END_IF

        _done := _plcCycleCounter >= 10;
        ProbeDoneWhen(_done);
        {endregion}
        {region "T699_OnStateChangeWhenChangingModes"}
    eTcoSequencerTests.OnStateChangeWhenChangingModes:
        IF NOT _arranged THEN
            _sut_A.TcoSequencerTest := eTcoSequencerTests.OnStateChangeWhenChangingModes;
            _sut_N.TcoSequencerTest := eTcoSequencerTests.OnStateChangeWhenChangingModes;
            _sut_A.SetCyclicMode(); //Set sequencer into the cyclic mode
            _sut_N.SetCyclicMode(); //Set sequencer into the cyclic mode
            _sut_A.SetSequenceAsChecked(); //Set sequence as checked, so no StepID uniqueness is performed on next sequence execution
            _sut_N.SetSequenceAsChecked(); //Set sequence as checked, so no StepID uniqueness is performed on next sequence execution
            _sut_A.SetNumberOfSteps(_totalStepNumber);
            _sut_N.SetNumberOfSteps(_totalStepNumber);
            _sut_A.TotalStepNumber := _totalStepNumber;
            _sut_N.TotalStepNumber := _totalStepNumber;
            _sut_A.SaveNumberOfStepsInSequence();
            _sut_N.SaveNumberOfStepsInSequence();
            _sut_A.CyclicCycles := _cyclicCycles;
            _sut_N.CyclicCycles := _cyclicCycles;
            _sut_A.StepInEvents := _stepInEvents;
            _sut_N.StepInEvents := _stepInEvents;
            _sut_A.SequenceCycles := 0;
            _sut_N.SequenceCycles := 0;
            _plcCycleCounter := 0;
            _arranged := TRUE;
            RETURN;
        END_IF

        IF NOT _done THEN
            _sut_A.SequenceRun := _plcCycleCounter;
            _sut_N.SequenceRun := _plcCycleCounter;
            _sut_A.Run();
            _sut_N.Run();
            _sut_A.SaveNumberOfStepsInSequence();
            _sut_N.SaveNumberOfStepsInSequence();
        END_IF

        _done := _plcCycleCounter >= 2 * _cyclicCycles + _stepInEvents + 1;
        ProbeDoneWhen(_done);
        {endregion}
END_CASE
END_METHOD

METHOD INTERNAL ReadOutCycleCounters
_startCycles := THIS^.StartCycleCount;
_endCycles := THIS^.EndCycleCount;
_myIdentity := THIS^.Identity;
END_METHOD

END_FUNCTION_BLOCK

// ---- Tests/TcoSequencer/PlcExecuted/TcoSequencerTestType.TcPOU
FUNCTION_BLOCK TcoSequencerTestType EXTENDS TcoCore._internals_TcoSequencer
VAR
    _runOneStep : BOOL;
    _runAllSteps : BOOL;
    _finishStep : BOOL;
    _stepId : INT;
    _enabled : BOOL;
    _stepDescription : STRING(254);
    _currentStepId : INT;
    _currentStepDescription : STRING(254);
    _myTcoChildState : TcoSequencerTestChildState(THIS^, eRestoreMode.None);
    _onCompleteStepCount : INT;
    _onSequenceCompleteCount : INT;
    _onSequencerErrorCount : ULINT;
    _onStateChangeCount : ULINT;
    _stateChangeFrom : INT;
    _stateChangeTo : INT;
    _callRestoreInOnStateChange : BOOL;
    _numberOfSteps : UINT;
    _previousNumberOfSteps : UINT;
    _tcoSequencerTest : eTcoSequencerTests;
    _totalStepNumber : UINT;
    _sequenceRun : ULINT;
    _reqStep : INT;
    _reqStepNotExists : INT;
    _initReqStepCycle : UINT;
    _postOpenRequestStepCycle : UINT;
    _preCloseRequestStepCycle : UINT;
    _restoreCycleCount : UINT;
    _cyclicCycles : UINT;
    _stepInEvents : UINT;
    _sequenceCycles : UINT;
END_VAR

METHOD _RequestStep
VAR_INPUT
    inRequestedStepId : INT;
END_VAR
THIS^.RequestStep(inRequestedStepId);
END_METHOD

METHOD _SequenceComplete
THIS^.CompleteSequence();
END_METHOD

METHOD INTERNAL _Step : BOOL
VAR_INPUT
    inStepId : INT;
    inEnabled : BOOL;
    inStepDescription : STRING(254);
END_VAR
_Step := SUPER^.Step(inStepID := inStepId, inEnabled := inEnabled, inStepDescription := inStepDescription);
END_METHOD

METHOD _StepBackward
THIS^.ModeController.StepBackward();
END_METHOD

METHOD _StepCompleteWhen
VAR_INPUT
    inCondition : BOOL;
END_VAR
THIS^.StepCompleteWhen(inCondition);
END_METHOD

METHOD _StepForward
THIS^.ModeController.StepForward();
END_METHOD

METHOD INTERNAL _StepIn
THIS^.ModeController.StepIn();
END_METHOD

PROPERTY CallRestoreInOnStateChange : BOOL
GET
CallRestoreInOnStateChange := _callRestoreInOnStateChange;
END_GET
SET
_callRestoreInOnStateChange := CallRestoreInOnStateChange;
END_SET
END_PROPERTY

{attribute 'TcRpcEnable'}
METHOD INTERNAL ChildHasAutoRestoreEnabled : BOOL
ChildHasAutoRestoreEnabled := THIS^._myTcoChildState.IsAutoRestoreEnabled;
END_METHOD

{attribute 'TcRpcEnable'}
METHOD INTERNAL ChildIsAutoRestorable : BOOL
ChildIsAutoRestorable := THIS^._myTcoChildState.AutoRestorable;
END_METHOD

METHOD INTERNAL ClearNumberOfSteps
_stepCounter := 0;
_numberOfStepsInSequence := 0;
_previousNumberOfStepsInSequence := 0;
END_METHOD

PROPERTY CyclicCycles : UINT
GET
CyclicCycles := _cyclicCycles;
END_GET
SET
_cyclicCycles := CyclicCycles;
END_SET
END_PROPERTY

PROPERTY Enabled : BOOL
GET
Enabled := _enabled;
END_GET
SET
_enabled := Enabled;
END_SET
END_PROPERTY

PROPERTY FinishStep : BOOL
GET
FinishStep := _finishStep;
END_GET
SET
_finishStep := FinishStep;
END_SET
END_PROPERTY

{attribute 'TcRpcEnable'}
METHOD INTERNAL GetChildState : INT
GetChildState := THIS^._myTcoChildState.State;
END_METHOD

{attribute 'TcRpcEnable'}
METHOD GetOrderOfTheCurrentlyEvaluatedStep : UINT
GetOrderOfTheCurrentlyEvaluatedStep := _theOrderOfTheCurrentlyEvaluatedStep;
END_METHOD

{attribute 'TcRpcEnable'}
METHOD GetOrderOfTheCurrentlyExecutedStep : UINT
GetOrderOfTheCurrentlyExecutedStep := _theOrderOfTheCurrentlyExecutedStep;
END_METHOD

{attribute 'TcRpcEnable'}
METHOD GetRequestStepCycle : UINT
GetRequestStepCycle := RequestStepCycle;
END_METHOD

{attribute 'TcRpcEnable'}
METHOD INTERNAL HasAutoRestoreEnabled : BOOL
HasAutoRestoreEnabled := SUPER^.IsAutoRestoreEnabled;
END_METHOD

PROPERTY InitReqStepCycle : UINT
GET
_initReqStepCycle := RequestStepCycle;
InitReqStepCycle := _initReqStepCycle;
END_GET
SET
_initReqStepCycle := InitReqStepCycle;
RequestStepCycle := _initReqStepCycle;
END_SET
END_PROPERTY

{attribute 'TcRpcEnable'}
METHOD INTERNAL IsAutoRestorable : BOOL
IsAutoRestorable := SUPER^.AutoRestorable;
END_METHOD

METHOD PROTECTED Main : BOOL
CASE _tcoSequencerTest OF
    eTcoSequencerTests.NumberOfStepsCount, eTcoSequencerTests.OnStateChangeWithRestoreCallInside:
        MAIN_NumberOfStepsCount();
    eTcoSequencerTests.ExecutionInOnePLCcycle, eTcoSequencerTests.OnStepCompleted, eTcoSequencerTests.OnSequenceCompleted:
        MAIN_ExecutionInOnePLCcycle();
    eTcoSequencerTests.RestoreChildBetweenSteps:
        MAIN_RestoreChildBetweenSteps();
    eTcoSequencerTests.MinStepId:
        MAIN_MinStepId();
    eTcoSequencerTests.MaxStepId:
        MAIN_MaxStepId();
    eTcoSequencerTests.RequestStepToFirstStepWithStepId0:
        MAIN_RequestStepToFirstStepWithStepId0();
    eTcoSequencerTests.RequestStep:
        MAIN_RequestStep();
    eTcoSequencerTests.CheckStepIdUniqueness, eTcoSequencerTests.RestoreAlreadyCheckedSequence, eTcoSequencerTests.NotUniqueStepId,
        eTcoSequencerTests.AfterErrorRestore, eTcoSequencerTests.CheckStepIdUniquenessStepMode, eTcoSequencerTests.NotUniqueStepIdInStepMode,
        eTcoSequencerTests.InvalidModeDetailed, eTcoSequencerTests.StepInErrorDetailed:
        MAIN_CheckStepIdUniqueness();
    eTcoSequencerTests.ChangeStepIdDuringExecution:
        MAIN_ChangeStepIdDuringExecution();
    eTcoSequencerTests.CommentOutPartOfRunningSequencer:
        MAIN_CommentOutPartOfRunningSequencer();
    eTcoSequencerTests.UncommentPartOfRunningSequencer:
        MAIN_UncommentPartOfRunningSequencer();
    eTcoSequencerTests.RequestStepFromLowerToHigher:
        MAIN_RequestStepFromLowerToHigher();
    eTcoSequencerTests.RequestStepFromHigherToLower:
        MAIN_RequestStepFromHigherToLower();
    eTcoSequencerTests.RequestStepToNotExistingStep, eTcoSequencerTests.StepModeRequestStepToNotExistingStep:
        MAIN_RequestStepToNotExistingStep();
    eTcoSequencerTests.RequestStepWhilePreviousRequestStepHasNotBeenYetProcessed,
        eTcoSequencerTests.StepModeRequestStepWhilePreviousRequestStepHasnotBeenYetProcessed:
        MAIN_RequestStepWhilePreviousRequestStepHasNotBeenYetProcessed();
    eTcoSequencerTests.SetStepMode:
        MAIN_SetStepMode();
    eTcoSequencerTests.StepMode:
        MAIN_StepMode();
    eTcoSequencerTests.StepModeStepIn:
        MAIN_StepModeStepIn();
    eTcoSequencerTests.StepModeChangeStepIdDuringExecution:
        MAIN_StepModeChangeStepIdDuringExecution();
    eTcoSequencerTests.StepModeChangeStepOrder:
        MAIN_StepModeChangeStepOrder();
    eTcoSequencerTests.StepModeCommentOutPartOfRunningSequencer:
        MAIN_StepModeCommentOutPartOfRunningSequencer();
    eTcoSequencerTests.StepModeUncommentPartOfRunningSequencer:
        MAIN_StepModeUncommentPartOfRunningSequencer();
    eTcoSequencerTests.StepModeRequestStepFromLowerToHigher:
        MAIN_StepModeRequestStepFromLowerToHigher();
    eTcoSequencerTests.StepModeRequestStepFromHigherToLower:
        MAIN_StepModeRequestStepFromHigherToLower();
    eTcoSequencerTests.StepModeDisabledStep:
        MAIN_StepModeDisabledStep();
    eTcoSequencerTests.StepModeStepForwardBackward:
        MAIN_StepModeStepForwardBackward();
    eTcoSequencerTests.StepModeStepInDetailed:
        MAIN_StepModeStepInDetailed();
    eTcoSequencerTests.SwitchStepModeOnDuringStepExecution:
        MAIN_SwitchStepModeOnDuringStepExecution();
    eTcoSequencerTests.StepModeStepForwardFromRunningStep:
        MAIN_StepModeStepForwardFromRunningStep();
    eTcoSequencerTests.StepModeStepBackwardFromRunningStep:
        MAIN_StepModeStepBackwardFromRunningStep();
    eTcoSequencerTests.SwitchStepModeStepOffFromReadyToRun:
        MAIN_SwitchStepModeStepOffFromReadyToRun();
    eTcoSequencerTests.SwitchStepModeStepOffFromRunning:
        MAIN_SwitchStepModeStepOffFromRunning();
    eTcoSequencerTests.SwitchStepModeStepOnFromRunning:
        MAIN_SwitchStepModeStepOnFromRunning();
    eTcoSequencerTests.OnStateChangeWhenChangingModes:
        MAIN_OnStateChangeWhenChangingModes();
END_CASE
END_METHOD

METHOD MAIN_ChangeStepIdDuringExecution
VAR
    i : INT;
END_VAR
IF _sequenceRun = 1 THEN
    IF Step(0, TRUE, 'Step number 0') THEN
        StepCompleteWhen(TRUE);
    END_IF

    FOR i := 1 TO _totalStepNumber - 2 DO
        IF Step(i, TRUE, CONCAT('Step ', INT_TO_STRING(i))) THEN
            StepCompleteWhen(FALSE);
        END_IF
    END_FOR

    IF Step(_totalStepNumber - 1, TRUE, CONCAT('Step ', INT_TO_STRING(_totalStepNumber - 1))) THEN
        _SequenceComplete();
    END_IF
END_IF

IF _sequenceRun = 2 THEN
    IF Step(0, TRUE, 'Step 0') THEN
        StepCompleteWhen(TRUE);
    END_IF

    IF Step(1, TRUE, 'Step 1') THEN
        StepCompleteWhen(TRUE);
    END_IF

    IF Step(2, TRUE, 'Step 2') THEN
        StepCompleteWhen(FALSE);
    END_IF

    IF Step(3, TRUE, 'Step 3') THEN
        StepCompleteWhen(FALSE);
    END_IF

    FOR i := 4 TO _totalStepNumber - 2 DO
        IF Step(i, TRUE, CONCAT('Step ', INT_TO_STRING(i))) THEN
            StepCompleteWhen(FALSE);
        END_IF
    END_FOR

    IF Step(_totalStepNumber - 1, TRUE, CONCAT('Step ', INT_TO_STRING(_totalStepNumber - 1))) THEN
        _SequenceComplete();
    END_IF
END_IF

IF _sequenceRun = 3 THEN
    IF Step(0, TRUE, 'Step 0') THEN
        StepCompleteWhen(TRUE);
    END_IF

    IF Step(1, TRUE, 'Step 1') THEN
        StepCompleteWhen(TRUE);
    END_IF

    IF Step(3, TRUE, 'Step 2') THEN
        StepCompleteWhen(FALSE);
    END_IF

    IF Step(2, TRUE, 'Step 3') THEN
        StepCompleteWhen(FALSE);
    END_IF

    FOR i := 4 TO _totalStepNumber - 2 DO
        IF Step(i, TRUE, CONCAT('Step ', INT_TO_STRING(i))) THEN
            StepCompleteWhen(FALSE);
        END_IF
    END_FOR

    IF Step(_totalStepNumber - 1, TRUE, CONCAT('Step ', INT_TO_STRING(_totalStepNumber - 1))) THEN
        _SequenceComplete();
    END_IF
END_IF
END_METHOD

METHOD MAIN_CheckStepIdUniqueness
//******************************************************************
IF SUPER^.Step(0, TRUE, 'Step number 0') THEN
    SUPER^.StepCompleteWhen((_runOneStep OR _runAllSteps) AND _finishStep);

    IF _runOneStep THEN
        _runOneStep := FALSE;
        RETURN;
    END_IF
END_IF

IF SUPER^.Step(1, TRUE, 'Step number 1') THEN
    SUPER^.StepCompleteWhen((_runOneStep OR _runAllSteps) AND _finishStep);

    IF _runOneStep THEN
        _runOneStep := FALSE;
        RETURN;
    END_IF
END_IF

IF SUPER^.Step(2, TRUE, 'Step number 2') THEN
    SUPER^.StepCompleteWhen((_runOneStep OR _runAllSteps) AND _finishStep);

    IF _runOneStep THEN
        _runOneStep := FALSE;
        RETURN;
    END_IF
END_IF

IF SUPER^.Step(3, TRUE, 'Step number 3') THEN
    SUPER^.StepCompleteWhen((_runOneStep OR _runAllSteps) AND _finishStep);

    IF _runOneStep THEN
        _runOneStep := FALSE;
        RETURN;
    END_IF
END_IF

IF SUPER^.Step(4, TRUE, 'Step number 4') THEN
    SUPER^.StepCompleteWhen((_runOneStep OR _runAllSteps) AND _finishStep);

    IF _runOneStep THEN
        _runOneStep := FALSE;
        RETURN;
    END_IF
END_IF

IF SUPER^.Step(5, TRUE, 'Step number 5') THEN
    SUPER^.StepCompleteWhen((_runOneStep OR _runAllSteps) AND _finishStep);

    IF _runOneStep THEN
        _runOneStep := FALSE;
        RETURN;
    END_IF
END_IF

IF SUPER^.Step(6, TRUE, 'Step number 6') THEN
    SUPER^.StepCompleteWhen((_runOneStep OR _runAllSteps) AND _finishStep);

    IF _runOneStep THEN
        _runOneStep := FALSE;
        RETURN;
    END_IF
END_IF

IF SUPER^.Step(7, TRUE, 'Step number 7') THEN
    SUPER^.StepCompleteWhen((_runOneStep OR _runAllSteps) AND _finishStep);

    IF _runOneStep THEN
        _runOneStep := FALSE;
        RETURN;
    END_IF
END_IF

IF SUPER^.Step(8, TRUE, 'Step number 8') THEN
    SUPER^.StepCompleteWhen((_runOneStep OR _runAllSteps) AND _finishStep);

    IF _runOneStep THEN
        _runOneStep := FALSE;
        RETURN;
    END_IF
END_IF

IF SUPER^.Step(9, TRUE, 'Step number 9') THEN
    SUPER^.StepCompleteWhen((_runOneStep OR _runAllSteps) AND _finishStep);

    IF _runOneStep THEN
        _runOneStep := FALSE;
        RETURN;
    END_IF
END_IF

IF SUPER^.Step(10, TRUE, 'Step number 10') THEN
    SUPER^.StepCompleteWhen((_runOneStep OR _runAllSteps) AND _finishStep);

    IF _runOneStep THEN
        _runOneStep := FALSE;
        RETURN;
    END_IF
END_IF

IF SUPER^.Step(11, TRUE, 'Step number 11') THEN
    SUPER^.StepCompleteWhen((_runOneStep OR _runAllSteps) AND _finishStep);

    IF _runOneStep THEN
        _runOneStep := FALSE;
        RETURN;
    END_IF
END_IF

IF SUPER^.Step(12, TRUE, 'Step number 12') THEN
    SUPER^.StepCompleteWhen((_runOneStep OR _runAllSteps) AND _finishStep);

    IF _runOneStep THEN
        _runOneStep := FALSE;
        RETURN;
    END_IF
END_IF

IF SUPER^.Step(13, TRUE, 'Step number 13') THEN
    SUPER^.StepCompleteWhen((_runOneStep OR _runAllSteps) AND _finishStep);

    IF _runOneStep THEN
        _runOneStep := FALSE;
        RETURN;
    END_IF
END_IF

IF SUPER^.Step(14, TRUE, 'Step number 14') THEN
    SUPER^.StepCompleteWhen((_runOneStep OR _runAllSteps) AND _finishStep);

    IF _runOneStep THEN
        _runOneStep := FALSE;
        RETURN;
    END_IF
END_IF

IF SUPER^.Step(15, TRUE, 'Step number 15') THEN
    SUPER^.StepCompleteWhen((_runOneStep OR _runAllSteps) AND _finishStep);

    IF _runOneStep THEN
        _runOneStep := FALSE;
        RETURN;
    END_IF
END_IF

IF SUPER^.Step(16, TRUE, 'Step number 16') THEN
    SUPER^.StepCompleteWhen((_runOneStep OR _runAllSteps) AND _finishStep);

    IF _runOneStep THEN
        _runOneStep := FALSE;
        RETURN;
    END_IF
END_IF

IF SUPER^.Step(17, TRUE, 'Step number 17') THEN
    SUPER^.StepCompleteWhen((_runOneStep OR _runAllSteps) AND _finishStep);

    IF _runOneStep THEN
        _runOneStep := FALSE;
        RETURN;
    END_IF
END_IF

IF SUPER^.Step(18, TRUE, 'Step number 18') THEN
    SUPER^.StepCompleteWhen((_runOneStep OR _runAllSteps) AND _finishStep);

    IF _runOneStep THEN
        _runOneStep := FALSE;
        RETURN;
    END_IF
END_IF

IF SUPER^.Step(19, TRUE, 'Step number 19') THEN
    SUPER^.StepCompleteWhen((_runOneStep OR _runAllSteps) AND _finishStep);

    IF _runOneStep THEN
        _runOneStep := FALSE;
        RETURN;
    END_IF
END_IF

IF SUPER^.Step(20, TRUE, 'Step number 20') THEN
    SUPER^.StepCompleteWhen((_runOneStep OR _runAllSteps) AND _finishStep);

    IF _runOneStep THEN
        _runOneStep := FALSE;
        RETURN;
    END_IF
END_IF

IF SUPER^.Step(21, TRUE, 'Step number 21') THEN
    SUPER^.StepCompleteWhen((_runOneStep OR _runAllSteps) AND _finishStep);

    IF _runOneStep THEN
        _runOneStep := FALSE;
        RETURN;
    END_IF
END_IF

IF SUPER^.Step(22, TRUE, 'Step number 22') THEN
    SUPER^.StepCompleteWhen((_runOneStep OR _runAllSteps) AND _finishStep);

    IF _runOneStep THEN
        _runOneStep := FALSE;
        RETURN;
    END_IF
END_IF

IF SUPER^.Step(23, TRUE, 'Step number 23') THEN
    SUPER^.StepCompleteWhen((_runOneStep OR _runAllSteps) AND _finishStep);

    IF _runOneStep THEN
        _runOneStep := FALSE;
        RETURN;
    END_IF
END_IF

IF SUPER^.Step(24, TRUE, 'Step number 24') THEN
    SUPER^.StepCompleteWhen((_runOneStep OR _runAllSteps) AND _finishStep);

    IF _runOneStep THEN
        _runOneStep := FALSE;
        RETURN;
    END_IF
END_IF

IF SUPER^.Step(25, TRUE, 'Step number 25') THEN
    SUPER^.StepCompleteWhen((_runOneStep OR _runAllSteps) AND _finishStep);

    IF _runOneStep THEN
        _runOneStep := FALSE;
        RETURN;
    END_IF
END_IF

IF SUPER^.Step(26, TRUE, 'Step number 26') THEN
    SUPER^.StepCompleteWhen((_runOneStep OR _runAllSteps) AND _finishStep);

    IF _runOneStep THEN
        _runOneStep := FALSE;
        RETURN;
    END_IF
END_IF

IF SUPER^.Step(27, TRUE, 'Step number 27') THEN
    SUPER^.StepCompleteWhen((_runOneStep OR _runAllSteps) AND _finishStep);

    IF _runOneStep THEN
        _runOneStep := FALSE;
        RETURN;
    END_IF
END_IF

IF SUPER^.Step(28, TRUE, 'Step number 28') THEN
    SUPER^.StepCompleteWhen((_runOneStep OR _runAllSteps) AND _finishStep);

    IF _runOneStep THEN
        _runOneStep := FALSE;
        RETURN;
    END_IF
END_IF

IF SUPER^.Step(29, TRUE, 'Step number 29') THEN
    SUPER^.StepCompleteWhen((_runOneStep OR _runAllSteps) AND _finishStep);

    IF _runOneStep THEN
        _runOneStep := FALSE;
        RETURN;
    END_IF
END_IF

IF SUPER^.Step(30, TRUE, 'Step number 30') THEN
    SUPER^.StepCompleteWhen((_runOneStep OR _runAllSteps) AND _finishStep);

    IF _runOneStep THEN
        _runOneStep := FALSE;
        RETURN;
    END_IF
END_IF

IF SUPER^.Step(31, TRUE, 'Step number 31') THEN
    SUPER^.StepCompleteWhen((_runOneStep OR _runAllSteps) AND _finishStep);

    IF _runOneStep THEN
        _runOneStep := FALSE;
        RETURN;
    END_IF
END_IF

IF SUPER^.Step(32, TRUE, 'Step number 32') THEN
    SUPER^.StepCompleteWhen((_runOneStep OR _runAllSteps) AND _finishStep);

    IF _runOneStep THEN
        _runOneStep := FALSE;
        RETURN;
    END_IF
END_IF

IF SUPER^.Step(33, TRUE, 'Step number 33') THEN
    SUPER^.StepCompleteWhen((_runOneStep OR _runAllSteps) AND _finishStep);

    IF _runOneStep THEN
        _runOneStep := FALSE;
        RETURN;
    END_IF
END_IF

IF SUPER^.Step(34, TRUE, 'Step number 34') THEN
    SUPER^.StepCompleteWhen((_runOneStep OR _runAllSteps) AND _finishStep);

    IF _runOneStep THEN
        _runOneStep := FALSE;
        RETURN;
    END_IF
END_IF

IF SUPER^.Step(35, TRUE, 'Step number 35') THEN
    SUPER^.StepCompleteWhen((_runOneStep OR _runAllSteps) AND _finishStep);

    IF _runOneStep THEN
        _runOneStep := FALSE;
        RETURN;
    END_IF
END_IF

IF SUPER^.Step(36, TRUE, 'Step number 36') THEN
    SUPER^.StepCompleteWhen((_runOneStep OR _runAllSteps) AND _finishStep);

    IF _runOneStep THEN
        _runOneStep := FALSE;
        RETURN;
    END_IF
END_IF

IF SUPER^.Step(37, TRUE, 'Step number 37') THEN
    SUPER^.StepCompleteWhen((_runOneStep OR _runAllSteps) AND _finishStep);

    IF _runOneStep THEN
        _runOneStep := FALSE;
        RETURN;
    END_IF
END_IF

IF SUPER^.Step(38, TRUE, 'Step number 38') THEN
    SUPER^.StepCompleteWhen((_runOneStep OR _runAllSteps) AND _finishStep);

    IF _runOneStep THEN
        _runOneStep := FALSE;
        RETURN;
    END_IF
END_IF

IF SUPER^.Step(39, TRUE, 'Step number 39') THEN
    SUPER^.StepCompleteWhen((_runOneStep OR _runAllSteps) AND _finishStep);

    IF _runOneStep THEN
        _runOneStep := FALSE;
        RETURN;
    END_IF
END_IF

IF SUPER^.Step(40, TRUE, 'Step number 40') THEN
    SUPER^.StepCompleteWhen((_runOneStep OR _runAllSteps) AND _finishStep);

    IF _runOneStep THEN
        _runOneStep := FALSE;
        RETURN;
    END_IF
END_IF

IF SUPER^.Step(41, TRUE, 'Step number 41') THEN
    SUPER^.StepCompleteWhen((_runOneStep OR _runAllSteps) AND _finishStep);

    IF _runOneStep THEN
        _runOneStep := FALSE;
        RETURN;
    END_IF
END_IF

IF SUPER^.Step(42, TRUE, 'Step number 42') THEN
    SUPER^.StepCompleteWhen((_runOneStep OR _runAllSteps) AND _finishStep);

    IF _runOneStep THEN
        _runOneStep := FALSE;
        RETURN;
    END_IF
END_IF

IF SUPER^.Step(43, TRUE, 'Step number 43') THEN
    SUPER^.StepCompleteWhen((_runOneStep OR _runAllSteps) AND _finishStep);

    IF _runOneStep THEN
        _runOneStep := FALSE;
        RETURN;
    END_IF
END_IF

IF SUPER^.Step(44, TRUE, 'Step number 44') THEN
    SUPER^.StepCompleteWhen((_runOneStep OR _runAllSteps) AND _finishStep);

    IF _runOneStep THEN
        _runOneStep := FALSE;
        RETURN;
    END_IF
END_IF

IF SUPER^.Step(45, TRUE, 'Step number 45') THEN
    SUPER^.StepCompleteWhen((_runOneStep OR _runAllSteps) AND _finishStep);

    IF _runOneStep THEN
        _runOneStep := FALSE;
        RETURN;
    END_IF
END_IF

IF SUPER^.Step(46, TRUE, 'Step number 46') THEN
    SUPER^.StepCompleteWhen((_runOneStep OR _runAllSteps) AND _finishStep);

    IF _runOneStep THEN
        _runOneStep := FALSE;
        RETURN;
    END_IF
END_IF

IF SUPER^.Step(47, TRUE, 'Step number 47') THEN
    SUPER^.StepCompleteWhen((_runOneStep OR _runAllSteps) AND _finishStep);

    IF _runOneStep THEN
        _runOneStep := FALSE;
        RETURN;
    END_IF
END_IF

IF SUPER^.Step(48, TRUE, 'Step number 48') THEN
    SUPER^.StepCompleteWhen((_runOneStep OR _runAllSteps) AND _finishStep);

    IF _runOneStep THEN
        _runOneStep := FALSE;
        RETURN;
    END_IF
END_IF

IF SUPER^.Step(49, TRUE, 'Step number 49') THEN
    SUPER^.StepCompleteWhen((_runOneStep OR _runAllSteps) AND _finishStep);

    IF _runOneStep THEN
        _runOneStep := FALSE;
        RETURN;
    END_IF
END_IF

IF SUPER^.Step(50, TRUE, 'Step number 50') THEN
    SUPER^.StepCompleteWhen((_runOneStep OR _runAllSteps) AND _finishStep);

    IF _runOneStep THEN
        _runOneStep := FALSE;
        RETURN;
    END_IF
END_IF

IF SUPER^.Step(51, TRUE, 'Step number 51') THEN
    SUPER^.StepCompleteWhen((_runOneStep OR _runAllSteps) AND _finishStep);

    IF _runOneStep THEN
        _runOneStep := FALSE;
        RETURN;
    END_IF
END_IF

IF SUPER^.Step(52, TRUE, 'Step number 52') THEN
    SUPER^.StepCompleteWhen((_runOneStep OR _runAllSteps) AND _finishStep);

    IF _runOneStep THEN
        _runOneStep := FALSE;
        RETURN;
    END_IF
END_IF

IF SUPER^.Step(53, TRUE, 'Step number 53') THEN
    SUPER^.StepCompleteWhen((_runOneStep OR _runAllSteps) AND _finishStep);

    IF _runOneStep THEN
        _runOneStep := FALSE;
        RETURN;
    END_IF
END_IF

IF SUPER^.Step(54, TRUE, 'Step number 54') THEN
    SUPER^.StepCompleteWhen((_runOneStep OR _runAllSteps) AND _finishStep);

    IF _runOneStep THEN
        _runOneStep := FALSE;
        RETURN;
    END_IF
END_IF

IF SUPER^.Step(55, TRUE, 'Step number 55') THEN
    SUPER^.StepCompleteWhen((_runOneStep OR _runAllSteps) AND _finishStep);

    IF _runOneStep THEN
        _runOneStep := FALSE;
        RETURN;
    END_IF
END_IF

IF SUPER^.Step(56, TRUE, 'Step number 56') THEN
    SUPER^.StepCompleteWhen((_runOneStep OR _runAllSteps) AND _finishStep);

    IF _runOneStep THEN
        _runOneStep := FALSE;
        RETURN;
    END_IF
END_IF

IF SUPER^.Step(57, TRUE, 'Step number 57') THEN
    SUPER^.StepCompleteWhen((_runOneStep OR _runAllSteps) AND _finishStep);

    IF _runOneStep THEN
        _runOneStep := FALSE;
        RETURN;
    END_IF
END_IF

IF SUPER^.Step(58, TRUE, 'Step number 58') THEN
    SUPER^.StepCompleteWhen((_runOneStep OR _runAllSteps) AND _finishStep);

    IF _runOneStep THEN
        _runOneStep := FALSE;
        RETURN;
    END_IF
END_IF

IF SUPER^.Step(59, TRUE, 'Step number 59') THEN
    SUPER^.StepCompleteWhen((_runOneStep OR _runAllSteps) AND _finishStep);

    IF _runOneStep THEN
        _runOneStep := FALSE;
        RETURN;
    END_IF
END_IF

IF SUPER^.Step(60, TRUE, 'Step number 60') THEN
    SUPER^.StepCompleteWhen((_runOneStep OR _runAllSteps) AND _finishStep);

    IF _runOneStep THEN
        _runOneStep := FALSE;
        RETURN;
    END_IF
END_IF

IF SUPER^.Step(61, TRUE, 'Step number 61') THEN
    SUPER^.StepCompleteWhen((_runOneStep OR _runAllSteps) AND _finishStep);

    IF _runOneStep THEN
        _runOneStep := FALSE;
        RETURN;
    END_IF
END_IF

IF SUPER^.Step(62, TRUE, 'Step number 62') THEN
    SUPER^.StepCompleteWhen((_runOneStep OR _runAllSteps) AND _finishStep);

    IF _runOneStep THEN
        _runOneStep := FALSE;
        RETURN;
    END_IF
END_IF

IF SUPER^.Step(63, TRUE, 'Step number 63') THEN
    SUPER^.StepCompleteWhen((_runOneStep OR _runAllSteps) AND _finishStep);

    IF _runOneStep THEN
        _runOneStep := FALSE;
        RETURN;
    END_IF
END_IF

IF SUPER^.Step(64, TRUE, 'Step number 64') THEN
    SUPER^.StepCompleteWhen((_runOneStep OR _runAllSteps) AND _finishStep);

    IF _runOneStep THEN
        _runOneStep := FALSE;
        RETURN;
    END_IF
END_IF

IF SUPER^.Step(65, TRUE, 'Step number 65') THEN
    SUPER^.StepCompleteWhen((_runOneStep OR _runAllSteps) AND _finishStep);

    IF _runOneStep THEN
        _runOneStep := FALSE;
        RETURN;
    END_IF
END_IF

IF SUPER^.Step(66, TRUE, 'Step number 66') THEN
    SUPER^.StepCompleteWhen((_runOneStep OR _runAllSteps) AND _finishStep);

    IF _runOneStep THEN
        _runOneStep := FALSE;
        RETURN;
    END_IF
END_IF

IF SUPER^.Step(67, TRUE, 'Step number 67') THEN
    SUPER^.StepCompleteWhen((_runOneStep OR _runAllSteps) AND _finishStep);

    IF _runOneStep THEN
        _runOneStep := FALSE;
        RETURN;
    END_IF
END_IF

IF SUPER^.Step(68, TRUE, 'Step number 68') THEN
    SUPER^.StepCompleteWhen((_runOneStep OR _runAllSteps) AND _finishStep);

    IF _runOneStep THEN
        _runOneStep := FALSE;
        RETURN;
    END_IF
END_IF

IF SUPER^.Step(69, TRUE, 'Step number 69') THEN
    SUPER^.StepCompleteWhen((_runOneStep OR _runAllSteps) AND _finishStep);

    IF _runOneStep THEN
        _runOneStep := FALSE;
        RETURN;
    END_IF
END_IF

IF SUPER^.Step(70, TRUE, 'Step number 70') THEN
    SUPER^.StepCompleteWhen((_runOneStep OR _runAllSteps) AND _finishStep);

    IF _runOneStep THEN
        _runOneStep := FALSE;
        RETURN;
    END_IF
END_IF

IF SUPER^.Step(71, TRUE, 'Step number 71') THEN
    SUPER^.StepCompleteWhen((_runOneStep OR _runAllSteps) AND _finishStep);

    IF _runOneStep THEN
        _runOneStep := FALSE;
        RETURN;
    END_IF
END_IF

IF SUPER^.Step(72, TRUE, 'Step number 72') THEN
    SUPER^.StepCompleteWhen((_runOneStep OR _runAllSteps) AND _finishStep);

    IF _runOneStep THEN
        _runOneStep := FALSE;
        RETURN;
    END_IF
END_IF

IF SUPER^.Step(73, TRUE, 'Step number 73') THEN
    SUPER^.StepCompleteWhen((_runOneStep OR _runAllSteps) AND _finishStep);

    IF _runOneStep THEN
        _runOneStep := FALSE;
        RETURN;
    END_IF
END_IF

IF SUPER^.Step(74, TRUE, 'Step number 74') THEN
    SUPER^.StepCompleteWhen((_runOneStep OR _runAllSteps) AND _finishStep);

    IF _runOneStep THEN
        _runOneStep := FALSE;
        RETURN;
    END_IF
END_IF

IF SUPER^.Step(75, TRUE, 'Step number 75') THEN
    SUPER^.StepCompleteWhen((_runOneStep OR _runAllSteps) AND _finishStep);

    IF _runOneStep THEN
        _runOneStep := FALSE;
        RETURN;
    END_IF
END_IF

IF SUPER^.Step(76, TRUE, 'Step number 76') THEN
    SUPER^.StepCompleteWhen((_runOneStep OR _runAllSteps) AND _finishStep);

    IF _runOneStep THEN
        _runOneStep := FALSE;
        RETURN;
    END_IF
END_IF

IF SUPER^.Step(77, TRUE, 'Step number 77') THEN
    SUPER^.StepCompleteWhen((_runOneStep OR _runAllSteps) AND _finishStep);

    IF _runOneStep THEN
        _runOneStep := FALSE;
        RETURN;
    END_IF
END_IF

IF SUPER^.Step(78, TRUE, 'Step number 78') THEN
    SUPER^.StepCompleteWhen((_runOneStep OR _runAllSteps) AND _finishStep);

    IF _runOneStep THEN
        _runOneStep := FALSE;
        RETURN;
    END_IF
END_IF

IF SUPER^.Step(79, TRUE, 'Step number 79') THEN
    SUPER^.StepCompleteWhen((_runOneStep OR _runAllSteps) AND _finishStep);

    IF _runOneStep THEN
        _runOneStep := FALSE;
        RETURN;
    END_IF
END_IF

IF SUPER^.Step(80, TRUE, 'Step number 80') THEN
    SUPER^.StepCompleteWhen((_runOneStep OR _runAllSteps) AND _finishStep);

    IF _runOneStep THEN
        _runOneStep := FALSE;
        RETURN;
    END_IF
END_IF

IF SUPER^.Step(81, TRUE, 'Step number 81') THEN
    SUPER^.StepCompleteWhen((_runOneStep OR _runAllSteps) AND _finishStep);

    IF _runOneStep THEN
        _runOneStep := FALSE;
        RETURN;
    END_IF
END_IF

IF SUPER^.Step(82, TRUE, 'Step number 82') THEN
    SUPER^.StepCompleteWhen((_runOneStep OR _runAllSteps) AND _finishStep);

    IF _runOneStep THEN
        _runOneStep := FALSE;
        RETURN;
    END_IF
END_IF

IF SUPER^.Step(83, TRUE, 'Step number 83') THEN
    SUPER^.StepCompleteWhen((_runOneStep OR _runAllSteps) AND _finishStep);

    IF _runOneStep THEN
        _runOneStep := FALSE;
        RETURN;
    END_IF
END_IF

IF SUPER^.Step(84, TRUE, 'Step number 84') THEN
    SUPER^.StepCompleteWhen((_runOneStep OR _runAllSteps) AND _finishStep);

    IF _runOneStep THEN
        _runOneStep := FALSE;
        RETURN;
    END_IF
END_IF

IF SUPER^.Step(85, TRUE, 'Step number 85') THEN
    SUPER^.StepCompleteWhen((_runOneStep OR _runAllSteps) AND _finishStep);

    IF _runOneStep THEN
        _runOneStep := FALSE;
        RETURN;
    END_IF
END_IF

IF SUPER^.Step(86, TRUE, 'Step number 86') THEN
    SUPER^.StepCompleteWhen((_runOneStep OR _runAllSteps) AND _finishStep);

    IF _runOneStep THEN
        _runOneStep := FALSE;
        RETURN;
    END_IF
END_IF

IF SUPER^.Step(87, TRUE, 'Step number 87') THEN
    SUPER^.StepCompleteWhen((_runOneStep OR _runAllSteps) AND _finishStep);

    IF _runOneStep THEN
        _runOneStep := FALSE;
        RETURN;
    END_IF
END_IF

IF SUPER^.Step(88, TRUE, 'Step number 88') THEN
    SUPER^.StepCompleteWhen((_runOneStep OR _runAllSteps) AND _finishStep);

    IF _runOneStep THEN
        _runOneStep := FALSE;
        RETURN;
    END_IF
END_IF

IF SUPER^.Step(89, TRUE, 'Step number 89') THEN
    SUPER^.StepCompleteWhen((_runOneStep OR _runAllSteps) AND _finishStep);

    IF _runOneStep THEN
        _runOneStep := FALSE;
        RETURN;
    END_IF
END_IF

IF SUPER^.Step(90, TRUE, 'Step number 90') THEN
    SUPER^.StepCompleteWhen((_runOneStep OR _runAllSteps) AND _finishStep);

    IF _runOneStep THEN
        _runOneStep := FALSE;
        RETURN;
    END_IF
END_IF

IF SUPER^.Step(91, TRUE, 'Step number 91') THEN
    SUPER^.StepCompleteWhen((_runOneStep OR _runAllSteps) AND _finishStep);

    IF _runOneStep THEN
        _runOneStep := FALSE;
        RETURN;
    END_IF
END_IF

IF SUPER^.Step(92, TRUE, 'Step number 92') THEN
    SUPER^.StepCompleteWhen((_runOneStep OR _runAllSteps) AND _finishStep);

    IF _runOneStep THEN
        _runOneStep := FALSE;
        RETURN;
    END_IF
END_IF

IF SUPER^.Step(93, TRUE, 'Step number 93') THEN
    SUPER^.StepCompleteWhen((_runOneStep OR _runAllSteps) AND _finishStep);

    IF _runOneStep THEN
        _runOneStep := FALSE;
        RETURN;
    END_IF
END_IF

IF SUPER^.Step(94, TRUE, 'Step number 94') THEN
    SUPER^.StepCompleteWhen((_runOneStep OR _runAllSteps) AND _finishStep);

    IF _runOneStep THEN
        _runOneStep := FALSE;
        RETURN;
    END_IF
END_IF

IF SUPER^.Step(95, TRUE, 'Step number 95') THEN
    SUPER^.StepCompleteWhen((_runOneStep OR _runAllSteps) AND _finishStep);

    IF _runOneStep THEN
        _runOneStep := FALSE;
        RETURN;
    END_IF
END_IF

IF SUPER^.Step(96, TRUE, 'Step number 96') THEN
    SUPER^.StepCompleteWhen((_runOneStep OR _runAllSteps) AND _finishStep);

    IF _runOneStep THEN
        _runOneStep := FALSE;
        RETURN;
    END_IF
END_IF

IF SUPER^.Step(97, TRUE, 'Step number 97') THEN
    SUPER^.StepCompleteWhen((_runOneStep OR _runAllSteps) AND _finishStep);

    IF _runOneStep THEN
        _runOneStep := FALSE;
        RETURN;
    END_IF
END_IF

IF SUPER^.Step(98, TRUE, 'Step number 98') THEN
    SUPER^.StepCompleteWhen((_runOneStep OR _runAllSteps) AND _finishStep);

    IF _runOneStep THEN
        _runOneStep := FALSE;
        RETURN;
    END_IF
END_IF

IF SUPER^.Step(99, TRUE, 'Step number 99') THEN
    SUPER^.StepCompleteWhen((_runOneStep OR _runAllSteps) AND _finishStep);

    IF _runOneStep THEN
        _runOneStep := FALSE;
        RETURN;
    END_IF
END_IF

IF SUPER^.Step(100, TRUE, 'Step number 100') THEN
    SUPER^.StepCompleteWhen((_runOneStep OR _runAllSteps) AND _finishStep);

    IF _runOneStep THEN
        _runOneStep := FALSE;
        RETURN;
    END_IF
END_IF

IF SUPER^.Step(101, TRUE, 'Step number 101') THEN
    SUPER^.StepCompleteWhen((_runOneStep OR _runAllSteps) AND _finishStep);

    IF _runOneStep THEN
        _runOneStep := FALSE;
        RETURN;
    END_IF
END_IF

IF SUPER^.Step(102, TRUE, 'Step number 102') THEN
    SUPER^.StepCompleteWhen((_runOneStep OR _runAllSteps) AND _finishStep);

    IF _runOneStep THEN
        _runOneStep := FALSE;
        RETURN;
    END_IF
END_IF

IF SUPER^.Step(103, TRUE, 'Step number 103') THEN
    SUPER^.StepCompleteWhen((_runOneStep OR _runAllSteps) AND _finishStep);

    IF _runOneStep THEN
        _runOneStep := FALSE;
        RETURN;
    END_IF
END_IF

IF SUPER^.Step(104, TRUE, 'Step number 104') THEN
    SUPER^.StepCompleteWhen((_runOneStep OR _runAllSteps) AND _finishStep);

    IF _runOneStep THEN
        _runOneStep := FALSE;
        RETURN;
    END_IF
END_IF

IF SUPER^.Step(105, TRUE, 'Step number 105') THEN
    SUPER^.StepCompleteWhen((_runOneStep OR _runAllSteps) AND _finishStep);

    IF _runOneStep THEN
        _runOneStep := FALSE;
        RETURN;
    END_IF
END_IF

IF SUPER^.Step(106, TRUE, 'Step number 106') THEN
    SUPER^.StepCompleteWhen((_runOneStep OR _runAllSteps) AND _finishStep);

    IF _runOneStep THEN
        _runOneStep := FALSE;
        RETURN;
    END_IF
END_IF

IF SUPER^.Step(107, TRUE, 'Step number 107') THEN
    SUPER^.StepCompleteWhen((_runOneStep OR _runAllSteps) AND _finishStep);

    IF _runOneStep THEN
        _runOneStep := FALSE;
        RETURN;
    END_IF
END_IF

IF SUPER^.Step(108, TRUE, 'Step number 108') THEN
    SUPER^.StepCompleteWhen((_runOneStep OR _runAllSteps) AND _finishStep);

    IF _runOneStep THEN
        _runOneStep := FALSE;
        RETURN;
    END_IF
END_IF

IF SUPER^.Step(109, TRUE, 'Step number 109') THEN
    SUPER^.StepCompleteWhen((_runOneStep OR _runAllSteps) AND _finishStep);

    IF _runOneStep THEN
        _runOneStep := FALSE;
        RETURN;
    END_IF
END_IF

IF SUPER^.Step(110, TRUE, 'Step number 110') THEN
    SUPER^.StepCompleteWhen((_runOneStep OR _runAllSteps) AND _finishStep);

    IF _runOneStep THEN
        _runOneStep := FALSE;
        RETURN;
    END_IF
END_IF

IF SUPER^.Step(111, TRUE, 'Step number 111') THEN
    SUPER^.StepCompleteWhen((_runOneStep OR _runAllSteps) AND _finishStep);

    IF _runOneStep THEN
        _runOneStep := FALSE;
        RETURN;
    END_IF
END_IF

IF SUPER^.Step(112, TRUE, 'Step number 112') THEN
    SUPER^.StepCompleteWhen((_runOneStep OR _runAllSteps) AND _finishStep);

    IF _runOneStep THEN
        _runOneStep := FALSE;
        RETURN;
    END_IF
END_IF

IF SUPER^.Step(113, TRUE, 'Step number 113') THEN
    SUPER^.StepCompleteWhen((_runOneStep OR _runAllSteps) AND _finishStep);

    IF _runOneStep THEN
        _runOneStep := FALSE;
        RETURN;
    END_IF
END_IF

IF SUPER^.Step(114, TRUE, 'Step number 114') THEN
    SUPER^.StepCompleteWhen((_runOneStep OR _runAllSteps) AND _finishStep);

    IF _runOneStep THEN
        _runOneStep := FALSE;
        RETURN;
    END_IF
END_IF

IF SUPER^.Step(115, TRUE, 'Step number 115') THEN
    SUPER^.StepCompleteWhen((_runOneStep OR _runAllSteps) AND _finishStep);

    IF _runOneStep THEN
        _runOneStep := FALSE;
        RETURN;
    END_IF
END_IF

IF SUPER^.Step(116, TRUE, 'Step number 116') THEN
    SUPER^.StepCompleteWhen((_runOneStep OR _runAllSteps) AND _finishStep);

    IF _runOneStep THEN
        _runOneStep := FALSE;
        RETURN;
    END_IF
END_IF

IF SUPER^.Step(117, TRUE, 'Step number 117') THEN
    SUPER^.StepCompleteWhen((_runOneStep OR _runAllSteps) AND _finishStep);

    IF _runOneStep THEN
        _runOneStep := FALSE;
        RETURN;
    END_IF
END_IF

IF SUPER^.Step(118, TRUE, 'Step number 118') THEN
    SUPER^.StepCompleteWhen((_runOneStep OR _runAllSteps) AND _finishStep);

    IF _runOneStep THEN
        _runOneStep := FALSE;
        RETURN;
    END_IF
END_IF

IF SUPER^.Step(119, TRUE, 'Step number 119') THEN
    SUPER^.StepCompleteWhen((_runOneStep OR _runAllSteps) AND _finishStep);

    IF _runOneStep THEN
        _runOneStep := FALSE;
        RETURN;
    END_IF
END_IF

IF SUPER^.Step(120, TRUE, 'Step number 120') THEN
    SUPER^.StepCompleteWhen((_runOneStep OR _runAllSteps) AND _finishStep);

    IF _runOneStep THEN
        _runOneStep := FALSE;
        RETURN;
    END_IF
END_IF

IF SUPER^.Step(121, TRUE, 'Step number 121') THEN
    SUPER^.StepCompleteWhen((_runOneStep OR _runAllSteps) AND _finishStep);

    IF _runOneStep THEN
        _runOneStep := FALSE;
        RETURN;
    END_IF
END_IF

IF SUPER^.Step(122, TRUE, 'Step number 122') THEN
    SUPER^.StepCompleteWhen((_runOneStep OR _runAllSteps) AND _finishStep);

    IF _runOneStep THEN
        _runOneStep := FALSE;
        RETURN;
    END_IF
END_IF

IF SUPER^.Step(123, TRUE, 'Step number 123') THEN
    SUPER^.StepCompleteWhen((_runOneStep OR _runAllSteps) AND _finishStep);

    IF _runOneStep THEN
        _runOneStep := FALSE;
        RETURN;
    END_IF
END_IF

IF SUPER^.Step(124, TRUE, 'Step number 124') THEN
    SUPER^.StepCompleteWhen((_runOneStep OR _runAllSteps) AND _finishStep);

    IF _runOneStep THEN
        _runOneStep := FALSE;
        RETURN;
    END_IF
END_IF

IF SUPER^.Step(125, TRUE, 'Step number 125') THEN
    SUPER^.StepCompleteWhen((_runOneStep OR _runAllSteps) AND _finishStep);

    IF _runOneStep THEN
        _runOneStep := FALSE;
        RETURN;
    END_IF
END_IF

IF SUPER^.Step(126, TRUE, 'Step number 126') THEN
    SUPER^.StepCompleteWhen((_runOneStep OR _runAllSteps) AND _finishStep);

    IF _runOneStep THEN
        _runOneStep := FALSE;
        RETURN;
    END_IF
END_IF

IF SUPER^.Step(127, TRUE, 'Step number 127') THEN
    SUPER^.StepCompleteWhen((_runOneStep OR _runAllSteps) AND _finishStep);

    IF _runOneStep THEN
        _runOneStep := FALSE;
        RETURN;
    END_IF
END_IF

IF SUPER^.Step(128, TRUE, 'Step number 128') THEN
    SUPER^.StepCompleteWhen((_runOneStep OR _runAllSteps) AND _finishStep);

    IF _runOneStep THEN
        _runOneStep := FALSE;
        RETURN;
    END_IF
END_IF

IF SUPER^.Step(129, TRUE, 'Step number 129') THEN
    SUPER^.StepCompleteWhen((_runOneStep OR _runAllSteps) AND _finishStep);

    IF _runOneStep THEN
        _runOneStep := FALSE;
        RETURN;
    END_IF
END_IF

IF SUPER^.Step(130, TRUE, 'Step number 130') THEN
    SUPER^.StepCompleteWhen((_runOneStep OR _runAllSteps) AND _finishStep);

    IF _runOneStep THEN
        _runOneStep := FALSE;
        RETURN;
    END_IF
END_IF

IF SUPER^.Step(131, TRUE, 'Step number 131') THEN
    SUPER^.StepCompleteWhen((_runOneStep OR _runAllSteps) AND _finishStep);

    IF _runOneStep THEN
        _runOneStep := FALSE;
        RETURN;
    END_IF
END_IF

IF SUPER^.Step(132, TRUE, 'Step number 132') THEN
    SUPER^.StepCompleteWhen((_runOneStep OR _runAllSteps) AND _finishStep);

    IF _runOneStep THEN
        _runOneStep := FALSE;
        RETURN;
    END_IF
END_IF

IF SUPER^.Step(133, TRUE, 'Step number 133') THEN
    SUPER^.StepCompleteWhen((_runOneStep OR _runAllSteps) AND _finishStep);

    IF _runOneStep THEN
        _runOneStep := FALSE;
        RETURN;
    END_IF
END_IF

IF SUPER^.Step(134, TRUE, 'Step number 134') THEN
    SUPER^.StepCompleteWhen((_runOneStep OR _runAllSteps) AND _finishStep);

    IF _runOneStep THEN
        _runOneStep := FALSE;
        RETURN;
    END_IF
END_IF

IF SUPER^.Step(135, TRUE, 'Step number 135') THEN
    SUPER^.StepCompleteWhen((_runOneStep OR _runAllSteps) AND _finishStep);

    IF _runOneStep THEN
        _runOneStep := FALSE;
        RETURN;
    END_IF
END_IF

IF SUPER^.Step(136, TRUE, 'Step number 136') THEN
    SUPER^.StepCompleteWhen((_runOneStep OR _runAllSteps) AND _finishStep);

    IF _runOneStep THEN
        _runOneStep := FALSE;
        RETURN;
    END_IF
END_IF

IF SUPER^.Step(137, TRUE, 'Step number 137') THEN
    SUPER^.StepCompleteWhen((_runOneStep OR _runAllSteps) AND _finishStep);

    IF _runOneStep THEN
        _runOneStep := FALSE;
        RETURN;
    END_IF
END_IF

IF SUPER^.Step(138, TRUE, 'Step number 138') THEN
    SUPER^.StepCompleteWhen((_runOneStep OR _runAllSteps) AND _finishStep);

    IF _runOneStep THEN
        _runOneStep := FALSE;
        RETURN;
    END_IF
END_IF

IF SUPER^.Step(139, TRUE, 'Step number 139') THEN
    SUPER^.StepCompleteWhen((_runOneStep OR _runAllSteps) AND _finishStep);

    IF _runOneStep THEN
        _runOneStep := FALSE;
        RETURN;
    END_IF
END_IF

IF SUPER^.Step(140, TRUE, 'Step number 140') THEN
    SUPER^.StepCompleteWhen((_runOneStep OR _runAllSteps) AND _finishStep);

    IF _runOneStep THEN
        _runOneStep := FALSE;
        RETURN;
    END_IF
END_IF

IF SUPER^.Step(141, TRUE, 'Step number 141') THEN
    SUPER^.StepCompleteWhen((_runOneStep OR _runAllSteps) AND _finishStep);

    IF _runOneStep THEN
        _runOneStep := FALSE;
        RETURN;
    END_IF
END_IF

IF SUPER^.Step(142, TRUE, 'Step number 142') THEN
    SUPER^.StepCompleteWhen((_runOneStep OR _runAllSteps) AND _finishStep);

    IF _runOneStep THEN
        _runOneStep := FALSE;
        RETURN;
    END_IF
END_IF

IF SUPER^.Step(143, TRUE, 'Step number 143') THEN
    SUPER^.StepCompleteWhen((_runOneStep OR _runAllSteps) AND _finishStep);

    IF _runOneStep THEN
        _runOneStep := FALSE;
        RETURN;
    END_IF
END_IF

IF SUPER^.Step(144, TRUE, 'Step number 144') THEN
    SUPER^.StepCompleteWhen((_runOneStep OR _runAllSteps) AND _finishStep);

    IF _runOneStep THEN
        _runOneStep := FALSE;
        RETURN;
    END_IF
END_IF

IF SUPER^.Step(145, TRUE, 'Step number 145') THEN
    SUPER^.StepCompleteWhen((_runOneStep OR _runAllSteps) AND _finishStep);

    IF _runOneStep THEN
        _runOneStep := FALSE;
        RETURN;
    END_IF
END_IF

IF SUPER^.Step(146, TRUE, 'Step number 146') THEN
    SUPER^.StepCompleteWhen((_runOneStep OR _runAllSteps) AND _finishStep);

    IF _runOneStep THEN
        _runOneStep := FALSE;
        RETURN;
    END_IF
END_IF

IF SUPER^.Step(147, TRUE, 'Step number 147') THEN
    SUPER^.StepCompleteWhen((_runOneStep OR _runAllSteps) AND _finishStep);

    IF _runOneStep THEN
        _runOneStep := FALSE;
        RETURN;
    END_IF
END_IF

IF SUPER^.Step(148, TRUE, 'Step number 148') THEN
    SUPER^.StepCompleteWhen((_runOneStep OR _runAllSteps) AND _finishStep);

    IF _runOneStep THEN
        _runOneStep := FALSE;
        RETURN;
    END_IF
END_IF

IF SUPER^.Step(149, TRUE, 'Step number 149') THEN
    SUPER^.StepCompleteWhen((_runOneStep OR _runAllSteps) AND _finishStep);

    IF _runOneStep THEN
        _runOneStep := FALSE;
        RETURN;
    END_IF
END_IF

